// TIA Portal V20 export
// export: Created 2025-12-01T14:57:35.378217Z, ExportSetting None, DisplayName Totally Integrated Automation Portal, DisplayVersion V20 Update 3, DisplayName TIA Portal Openness, DisplayVersion V20 Update 3, DisplayName TIA Portal Version Control Interface, DisplayVersion V20 Update 3, DisplayName STEP 7 Professional, DisplayVersion V20 Update 3, DisplayName STEP 7 Safety, DisplayVersion V20 Update 2, DisplayName WinCC Basic/Comfort/Advanced, DisplayVersion V20 Update 3, DisplayName WinCC Professional, DisplayVersion V20 Update 3, DisplayName WinCC Unified, DisplayVersion V20 Update 3
FUNCTION_BLOCK "FB532_Ordenes_ELEV / VTD_V2"   // FB532, LAD
{ S7_Optimized_Access := 'FALSE' }
// stored: AutoNumber false, SetENOAutomatically false
   VAR_INPUT
      Estado_CBx : "EstadoZona";   // Estado de la Zona
      Maquina { ExternalVisible := 'False'; ExternalWritable := 'False'} : UInt;   // Numero de Máquina
      OrdenDesCarga_OK : Bool;
      Error_Tx : Bool;
   END_VAR
   VAR_OUTPUT
      PosicionDestino : Real;
      Orden : Bool;
   END_VAR
   VAR
      OrdenH01_TipoMovi { ExternalAccessible := 'False'; ExternalVisible := 'False'; ExternalWritable := 'False'; S7_SetPoint := 'True'} : "UDT_VTD_Orden";   // Tipo de Movimiento a Ejecutar con la Horquilla 1
      OrdenH02_TipoMovi { ExternalAccessible := 'False'; ExternalVisible := 'False'; ExternalWritable := 'False'; S7_SetPoint := 'True'} : "UDT_VTD_Orden";   // Tipo de Movimiento a Ejecutar con la Horquilla 2
      OrdenEnCurso : Struct
         EnH01_Poscicion : Real;
         EnH02_Poscicion : Real;
         EnH01_MesaCarga : UInt;
         EnH02_MesaCarga : UInt;
         EnH01_MesaDesCarga : UInt;
         EnH02_MesaDesCarga : UInt;
         EnH01_Existe : Bool;
         EnH02_Existe : Bool;
      END_STRUCT;
      OrdenJdT { ExternalAccessible := 'False'; ExternalVisible := 'False'; ExternalWritable := 'False'} : Struct
         Operacion : UInt;
         MesaHorquilla : UInt;
         MesaCargaDesCarga : UInt;
         VarMesaHorquilla : UInt;
         VarMesaCargaDesCarga : UInt;
         OrdenPoscionado_NOK : Bool;
      END_STRUCT;
      OrdenHMI : Struct
         MesaHorquilla { ExternalAccessible := 'False'; ExternalVisible := 'False'; ExternalWritable := 'False'} : UInt;
         MesaDestino { ExternalAccessible := 'False'; ExternalVisible := 'False'; ExternalWritable := 'False'} : UInt;
         VarMesaHorquilla { ExternalAccessible := 'False'; ExternalVisible := 'False'; ExternalWritable := 'False'} : UInt;
         VarMesaDestino { ExternalAccessible := 'False'; ExternalVisible := 'False'; ExternalWritable := 'False'} : UInt;
      END_STRUCT;
      MemoFlancos { ExternalAccessible := 'False'; ExternalVisible := 'False'; ExternalWritable := 'False'} : Struct
         H1 : Struct
            Posicionar : Bool;
            Carga_E1 : Bool;
            Carga_E2 : Bool;
            Carga_E3 : Bool;
            Carga_E4 : Bool;
            DesCarga_S1 : Bool;
            DesCarga_S2 : Bool;
            DesCarga_S3 : Bool;
            DesCarga_S4 : Bool;
         END_STRUCT;
         H2 : Struct
            Posicionar : Bool;
            Carga_E1 : Bool;
            Carga_E2 : Bool;
            Carga_E3 : Bool;
            Carga_E4 : Bool;
            DesCarga_S1 : Bool;
            DesCarga_S2 : Bool;
            DesCarga_S3 : Bool;
            DesCarga_S4 : Bool;
         END_STRUCT;
      END_STRUCT;
      Peticion : Struct
         Posicion : Real;
         Activa { ExternalAccessible := 'False'; ExternalVisible := 'False'; ExternalWritable := 'False'} : Bool;
      END_STRUCT;
      MesaCargaH01_OK : Bool;
      MesaDesCargaH01_OK : Bool;
      MesaCargaH02_OK : Bool;
      MesaDesCargaH02_OK : Bool;
   END_VAR
   VAR_TEMP
      EstadoVI_VTD : "EstadoMaquina";
      EstadoVI_MesaH1 : "EstadosMesa";   // Estado VI de la Mesa de la H01
      EstadoVI_MesaH2 : "EstadosMesa";   // Estado VI de la Mesa de la H02
      VarUTs : Struct
         PrimeraUT_EnMesa : UInt;
         MesaDestino : UInt;
      END_STRUCT;
      VarBusqueda : Struct
         Posicion : Real;
         Destino : UInt;
         Indice : UInt;
      END_STRUCT;
      VarInterlock : Struct
         Posicion : Real;
         Indice : UInt;
      END_STRUCT;
      NumVTD : UInt;
      NumMesaH1 : UInt;
      NumMesaH2 : UInt;
      Cero : Byte;
      ValorReturn : Int;
      EnMarchaVTDC : Bool;
   END_VAR
   VAR_TEMP   // added for the SCL form of the ladder/FBD networks
      _w1 : Bool;
      _w2 : Bool;
   END_VAR
BEGIN

REGION Network 1 (SCL): Inicializacion
   /////////////////////////////////////////////////////////////////////////////
   // --- Inicializar las Variables
   #Cero := 0;


   /////////////////////////////////////////////////////////////////////////////
   // --- Inicializar Variables En Horquilla 01
   IF #OrdenEnCurso.EnH01_Existe = FALSE THEN
       #ValorReturn := FILL(BVAL := #Cero, BLK => #OrdenH01_TipoMovi);
       #OrdenEnCurso.EnH01_Poscicion := 0.0;
       #OrdenEnCurso.EnH01_MesaCarga := 0;
       #OrdenEnCurso.EnH01_MesaDesCarga := 0;

   END_IF;


   /////////////////////////////////////////////////////////////////////////////
   // --- Inicializar Variables En Horquilla 01
   IF #OrdenEnCurso.EnH02_Existe = FALSE THEN
       #ValorReturn := FILL(BVAL := #Cero, BLK => #OrdenH02_TipoMovi);
       #OrdenEnCurso.EnH02_Poscicion := 0.0;
       #OrdenEnCurso.EnH02_MesaCarga := 0;
       #OrdenEnCurso.EnH02_MesaDesCarga := 0;

   END_IF;
END_REGION

REGION Network 2: ---- En Marcha VTDC
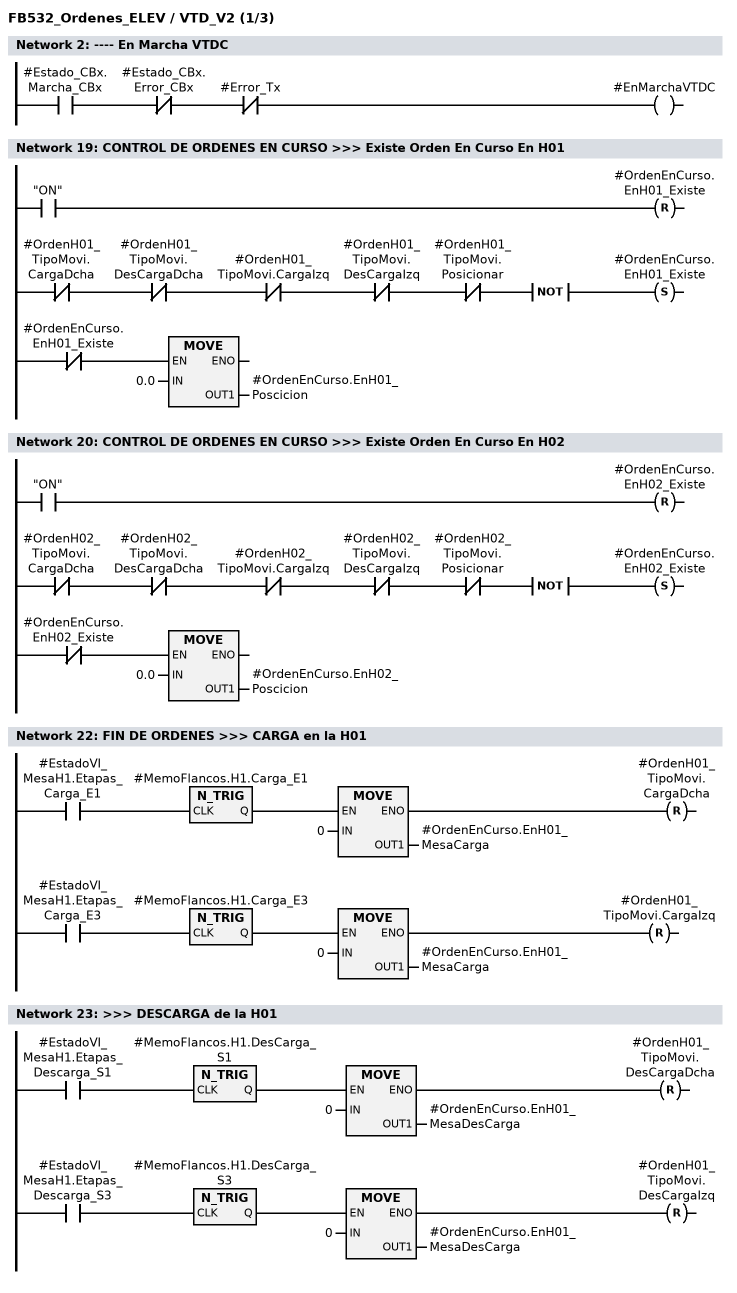
   RUNG wire#powerrail
      Contact( #Estado_CBx.Marcha_CBx )
      I_Contact( #Estado_CBx.Error_CBx )
      I_Contact( #Error_Tx )
      Coil( #EnMarchaVTDC )
   END_RUNG
   // the same network as SCL:
   #EnMarchaVTDC := #Estado_CBx.Marcha_CBx AND NOT #Estado_CBx.Error_CBx AND NOT #Error_Tx;
END_REGION

REGION Network 3 (SCL): ---- Recoger datos de la Maquina
   /////////////////////////////////////////////////////////////////////////////
   // Configuracion 
   #NumMesaH1 := #NumVTD := "DB885_ConfigMaquinas".Maquina[#Maquina].Mesa_1;
   #NumMesaH2 := "DB885_ConfigMaquinas".Maquina[#Maquina].Mesa_2;


   /////////////////////////////////////////////////////////////////////////////
   // Recoger ordenes de JdT
   #OrdenJdT.Operacion := "DB832_Maquinas".Maquinas[#NumVTD].VTD_ELEV.Operacion;
   #OrdenJdT.MesaHorquilla := "DB832_Maquinas".Maquinas[#NumVTD].VTD_ELEV.MesaHorquilla;
   #OrdenJdT.MesaCargaDesCarga := "DB832_Maquinas".Maquinas[#NumVTD].VTD_ELEV.MesaCargaDesCarga;
END_REGION

REGION Network 4 (SCL): ---- Recoger Estado VI de las Horquillas
   /////////////////////////////////////////////////////////////////////////////
   // - Recoger Estado de las Horquillas
   #EstadoVI_VTD := "DB904_Estado_Maquinas".EstadoVI[#NumVTD];
   #EstadoVI_MesaH1 := "DB900_Estado_Mesas".EstadoVI[#NumMesaH1];
   IF #NumMesaH2 <> 0 THEN
       #EstadoVI_MesaH2 := "DB900_Estado_Mesas".EstadoVI[#NumMesaH2];
   ELSE
       #ValorReturn := FILL(BVAL := #Cero, BLK => #EstadoVI_MesaH2);
   END_IF;
END_REGION

REGION Network 5 (SCL): ---- Recoger Variables Internas de las Horquillas
   /////////////////////////////////////////////////////////////////////////////
   // Recoger Variables para la Horquillla 01
   // OrdenDesCarga_OK >>> Permiso para Generar Orden de DesCarga, por si hay que hacer algun Calculo Previo de la Posicion
   #MesaCargaH01_OK := (#EstadoVI_MesaH1.Etapa_Vacia = TRUE) OR (#EstadoVI_MesaH1.Etapas_Descarga_S1 = TRUE) OR (#EstadoVI_MesaH1.Etapas_Descarga_S3 = TRUE);
   #MesaDesCargaH01_OK := (#EstadoVI_MesaH1.Etapa_Cargada = TRUE) AND (#OrdenDesCarga_OK = TRUE);


   /////////////////////////////////////////////////////////////////////////////
   /////////////////////////////////////////////////////////////////////////////
   // Recoger Variables para la Horquillla 02
   IF (#NumMesaH2 <> 0) THEN
       #MesaCargaH02_OK := (#EstadoVI_MesaH2.Etapa_Vacia = TRUE) OR (#EstadoVI_MesaH2.Etapas_Descarga_S1 = TRUE) OR (#EstadoVI_MesaH2.Etapas_Descarga_S3 = TRUE);
       #MesaDesCargaH02_OK := (#EstadoVI_MesaH2.Etapa_Cargada = TRUE);

   ELSE
       #MesaCargaH02_OK := #MesaDesCargaH02_OK = FALSE;

   END_IF;
END_REGION

REGION Network 6 (SCL): ---- Reset de Variables
   /////////////////////////////////////////////////////////////////////////////
   // Reseteo desde JdT
   IF #Estado_CBx.PerReset_CBx = TRUE THEN
       #Peticion.Activa := FALSE;
       #ValorReturn := FILL(BVAL := #Cero, BLK => #OrdenH01_TipoMovi);
       #ValorReturn := FILL(BVAL := #Cero, BLK => #OrdenH02_TipoMovi);

       #OrdenEnCurso.EnH01_Existe := #OrdenEnCurso.EnH02_Existe := FALSE;
       #OrdenEnCurso.EnH01_Poscicion := #OrdenEnCurso.EnH02_Poscicion := 0.0;
       #OrdenEnCurso.EnH01_MesaCarga := #OrdenEnCurso.EnH02_MesaCarga := 0;
       #OrdenEnCurso.EnH01_MesaDesCarga := #OrdenEnCurso.EnH02_MesaDesCarga := 0;

       #Peticion.Activa := FALSE;

   END_IF;
END_REGION

REGION Network 7: >>>>>>>>>>>>>>>>>>>>>>>>>>>>>>>>>>>>>>>>>>>>>>>>>>>>>>>>>>>>>>>>>>>>>>>>>>>>>>>>
END_REGION

REGION Network 8 (SCL): VTDC Doble (Particular del Tipo de Maquina) - Control H01 >>> CARGA
   /////////////////////////////////////////////////////////////////////////////
   // --- CONTROL DE CARGA de la Horquilla 01
   // 
   // --- Esta en Marcha 
   // --- Esta Preparado para Cargar
   // --- Comprobar que no exista Orden En Curso De Carga 
   IF (#EnMarchaVTDC = TRUE) AND (#MesaCargaH01_OK = TRUE) AND
       (#OrdenH01_TipoMovi.CargaDcha = FALSE) AND (#OrdenH01_TipoMovi.CargaIzq = FALSE) AND (#OrdenH01_TipoMovi.Posicionar = FALSE) THEN

       // >>>>> Sin Orden en Curso en la Horquilla 1
       //       Sin Orden En Curso en la Horquilla 2
       IF (#OrdenEnCurso.EnH01_Existe = FALSE) AND (#OrdenEnCurso.EnH02_Existe = FALSE) AND (#Peticion.Posicion = 0) THEN

           FOR #VarBusqueda.Indice := 1 TO "CTE_MaxMesas" DO
               // --- Hay Aviso de Entrada ???
               IF ("DB951_InterlockMaquinas".Maquina[#Maquina].Mesa[#VarBusqueda.Indice].Out.AVTF = TRUE) THEN

                   ////////////////////////////////////////////////////////////////////////////////
                   // --- Es Destino la Horquilla
                   #VarUTs.PrimeraUT_EnMesa := "DB810_ColasMesas".Colas[#VarBusqueda.Indice].UT_PrimeraMesa;
                   #VarBusqueda.Destino := "DB812_UTs_Control".UT[#VarUTs.PrimeraUT_EnMesa].MesaDestino;
                   #VarBusqueda.Destino := #VarBusqueda.Destino - "CTE_OffsetMesa";
                   IF (#VarBusqueda.Destino = #NumMesaH1) THEN
                       ////////////////////////////////////////////////////////////////////////////////
                       // --- Es En Carga Derecha
                       IF "DB885_ConfigMaquinas".Maquina[#Maquina].Mesa[#VarBusqueda.Indice].Derecha = TRUE THEN
                           #OrdenEnCurso.EnH01_Poscicion := "DB885_ConfigMaquinas".Maquina[#Maquina].Mesa[#VarBusqueda.Indice].Posicion_mm_H1;
                           #OrdenEnCurso.EnH01_MesaCarga := #VarBusqueda.Indice;
                           #OrdenH01_TipoMovi.CargaDcha := TRUE;
                           #OrdenEnCurso.EnH01_Existe := TRUE;
                           EXIT;
                       END_IF;
                       ////////////////////////////////////////////////////////////////////////////////
                       // --- Es En Carga Izquierda
                       IF "DB885_ConfigMaquinas".Maquina[#Maquina].Mesa[#VarBusqueda.Indice].Izquierda = TRUE THEN
                           #OrdenEnCurso.EnH01_Poscicion := "DB885_ConfigMaquinas".Maquina[#Maquina].Mesa[#VarBusqueda.Indice].Posicion_mm_H1;
                           #OrdenEnCurso.EnH01_MesaCarga := #VarBusqueda.Indice;
                           #OrdenH01_TipoMovi.CargaIzq := TRUE;
                           #OrdenEnCurso.EnH01_Existe := TRUE;
                           EXIT;
                       END_IF;
                   END_IF;
                   ////////////////////////////////////////////////////////////////////////////////

               END_IF;
           END_FOR;

       END_IF;


       // >>>>> Sin Orden en Curso en la Horquilla 1
       //       Con Orden En Curso en la Horquilla 2
       IF #OrdenEnCurso.EnH01_Existe = FALSE AND #OrdenEnCurso.EnH02_Existe = TRUE THEN
           #VarBusqueda.Posicion := #Peticion.Posicion;

           FOR #VarBusqueda.Indice := 1 TO "CTE_MaxMesas" DO
               // --- Hay Aviso de Entrada ???
               IF ("DB951_InterlockMaquinas".Maquina[#Maquina].Mesa[#VarBusqueda.Indice].Out.AVTF = TRUE) AND
                   ("DB885_ConfigMaquinas".Maquina[#Maquina].Mesa[#VarBusqueda.Indice].Posicion_mm_H1 = #VarBusqueda.Posicion) THEN

                   ////////////////////////////////////////////////////////////////////////////////
                   // --- Es Destino la Horquilla
                   #VarUTs.PrimeraUT_EnMesa := "DB810_ColasMesas".Colas[#VarBusqueda.Indice].UT_PrimeraMesa;
                   #VarBusqueda.Destino := "DB812_UTs_Control".UT[#VarUTs.PrimeraUT_EnMesa].MesaDestino;
                   #VarBusqueda.Destino := #VarBusqueda.Destino - "CTE_OffsetMesa";
                   IF (#VarBusqueda.Destino = #NumMesaH1) THEN
                       ////////////////////////////////////////////////////////////////////////////////
                       // --- Es En Carga Derecha
                       IF ("DB885_ConfigMaquinas".Maquina[#Maquina].Mesa[#VarBusqueda.Indice].Derecha = TRUE) THEN
                           #OrdenEnCurso.EnH01_Poscicion := "DB885_ConfigMaquinas".Maquina[#Maquina].Mesa[#VarBusqueda.Indice].Posicion_mm_H1;
                           #OrdenEnCurso.EnH01_MesaCarga := #VarBusqueda.Indice;
                           #OrdenH01_TipoMovi.CargaDcha := TRUE;
                           #OrdenEnCurso.EnH01_Existe := TRUE;
                           EXIT;
                       END_IF;
                       ////////////////////////////////////////////////////////////////////////////////
                       // --- Es En Carga Izquierda
                       IF ("DB885_ConfigMaquinas".Maquina[#Maquina].Mesa[#VarBusqueda.Indice].Izquierda = TRUE) THEN
                           #OrdenEnCurso.EnH01_Poscicion := "DB885_ConfigMaquinas".Maquina[#Maquina].Mesa[#VarBusqueda.Indice].Posicion_mm_H1;
                           #OrdenEnCurso.EnH01_MesaCarga := #VarBusqueda.Indice;
                           #OrdenH01_TipoMovi.CargaIzq := TRUE;
                           #OrdenEnCurso.EnH01_Existe := TRUE;
                           EXIT;
                       END_IF;
                   END_IF;
                   ////////////////////////////////////////////////////////////////////////////////

               END_IF;
           END_FOR;

       END_IF;


       // >>>>> Con Orden en Curso en la Horquilla 1
       //       Sin o Con Orden En Curso en la Horquilla 2
       IF #OrdenEnCurso.EnH01_Existe = TRUE THEN
           #VarBusqueda.Posicion := #Peticion.Posicion;

           FOR #VarBusqueda.Indice := 1 TO "CTE_MaxMesas" DO
               // --- Hay Aviso de Entrada ???
               IF ("DB951_InterlockMaquinas".Maquina[#Maquina].Mesa[#VarBusqueda.Indice].Out.AVTF = TRUE) AND
                   ("DB885_ConfigMaquinas".Maquina[#Maquina].Mesa[#VarBusqueda.Indice].Posicion_mm_H1 = #VarBusqueda.Posicion) THEN

                   ////////////////////////////////////////////////////////////////////////////////
                   // --- Es Destino la Horquilla
                   #VarUTs.PrimeraUT_EnMesa := "DB810_ColasMesas".Colas[#VarBusqueda.Indice].UT_PrimeraMesa;
                   #VarBusqueda.Destino := "DB812_UTs_Control".UT[#VarUTs.PrimeraUT_EnMesa].MesaDestino;
                   #VarBusqueda.Destino := #VarBusqueda.Destino - "CTE_OffsetMesa";
                   IF (#VarBusqueda.Destino = #NumMesaH1) THEN
                       ////////////////////////////////////////////////////////////////////////////////
                       // --- Es En Carga Derecha
                       IF ("DB885_ConfigMaquinas".Maquina[#Maquina].Mesa[#VarBusqueda.Indice].Derecha = TRUE) AND (#OrdenH01_TipoMovi.DesCargaIzq = TRUE) THEN
                           #OrdenEnCurso.EnH01_Poscicion := "DB885_ConfigMaquinas".Maquina[#Maquina].Mesa[#VarBusqueda.Indice].Posicion_mm_H1;
                           #OrdenEnCurso.EnH01_MesaCarga := #VarBusqueda.Indice;
                           #OrdenH01_TipoMovi.CargaDcha := TRUE;
                           #OrdenEnCurso.EnH01_Existe := TRUE;
                           EXIT;
                       END_IF;
                       ////////////////////////////////////////////////////////////////////////////////
                       // --- Es En Carga Izquierda
                       IF ("DB885_ConfigMaquinas".Maquina[#Maquina].Mesa[#VarBusqueda.Indice].Izquierda = TRUE) AND (#OrdenH01_TipoMovi.DesCargaDcha = TRUE) THEN
                           #OrdenEnCurso.EnH01_Poscicion := "DB885_ConfigMaquinas".Maquina[#Maquina].Mesa[#VarBusqueda.Indice].Posicion_mm_H1;
                           #OrdenEnCurso.EnH01_MesaCarga := #VarBusqueda.Indice;
                           #OrdenH01_TipoMovi.CargaIzq := TRUE;
                           #OrdenEnCurso.EnH01_Existe := TRUE;
                           EXIT;
                       END_IF;
                   END_IF;
                   ////////////////////////////////////////////////////////////////////////////////

               END_IF;
           END_FOR;

       END_IF;

   END_IF;
END_REGION

REGION Network 9 (SCL): VTDC Doble (Particular del Tipo de Maquina) - Control H01 >>> DESCARGA
   /////////////////////////////////////////////////////////////////////////////
   // --- CONTROL DE DESCARGA de la Horquilla 01
   // 
   // --- Esta en Marcha 
   // --- Esta Preparado para Cargar
   // --- Comprobar que no exista Orden En Curso De DesCarga 
   IF (#EnMarchaVTDC = TRUE) AND (#MesaDesCargaH01_OK = TRUE) AND
       (#OrdenH01_TipoMovi.DesCargaDcha = FALSE) AND (#OrdenH01_TipoMovi.DesCargaIzq = FALSE) AND (#OrdenH01_TipoMovi.Posicionar = FALSE) THEN

       /////////////////////////////////////////////////////////////////////////////
       // --- Recoger Destino de UT 
       #VarUTs.MesaDestino := 0;
       #VarUTs.PrimeraUT_EnMesa := "DB810_ColasMesas".Colas[#NumMesaH1].UT_PrimeraMesa;
       IF #VarUTs.PrimeraUT_EnMesa <> 0 THEN
           #VarUTs.MesaDestino := "DB812_UTs_Control".UT[#VarUTs.PrimeraUT_EnMesa].MesaDestino;
           IF (#VarUTs.MesaDestino <> 0) THEN
               #VarUTs.MesaDestino := #VarUTs.MesaDestino - "CTE_OffsetMesa";
               IF (#VarUTs.MesaDestino = #NumMesaH1) THEN
                   #VarUTs.MesaDestino := 0;
               END_IF;
           END_IF;

       END_IF;

       /////////////////////////////////////////////////////////////////////////////
       // --- Existe Destino de Salida
       IF #VarUTs.MesaDestino <> 0 THEN

           /////////////////////////////////////////////////////////////////////////////
           // >>>>> Sin Orden en Curso en la Horquilla 1
           //       Sin Orden En Curso en la Horquilla 2
           IF (#OrdenEnCurso.EnH01_Existe = FALSE) AND (#OrdenEnCurso.EnH02_Existe = FALSE) AND (#Peticion.Posicion = 0) THEN

               ////////////////////////////////////////////////////////////////////////////////
               // --- Es En DesCarga Derecha
               IF ("DB885_ConfigMaquinas".Maquina[#Maquina].Mesa[#VarUTs.MesaDestino].Derecha = TRUE) THEN
                   #OrdenEnCurso.EnH01_Poscicion := "DB885_ConfigMaquinas".Maquina[#Maquina].Mesa[#VarUTs.MesaDestino].Posicion_mm_H1;
                   #OrdenEnCurso.EnH01_MesaDesCarga := #VarUTs.MesaDestino;
                   #OrdenH01_TipoMovi.DesCargaDcha := TRUE;
                   #OrdenEnCurso.EnH01_Existe := TRUE;

               END_IF;
               ////////////////////////////////////////////////////////////////////////////////
               // --- Es En DesCarga Izquierda
               IF ("DB885_ConfigMaquinas".Maquina[#Maquina].Mesa[#VarUTs.MesaDestino].Izquierda = TRUE) THEN
                   #OrdenEnCurso.EnH01_Poscicion := "DB885_ConfigMaquinas".Maquina[#Maquina].Mesa[#VarUTs.MesaDestino].Posicion_mm_H1;
                   #OrdenEnCurso.EnH01_MesaDesCarga := #VarUTs.MesaDestino;
                   #OrdenH01_TipoMovi.DesCargaIzq := TRUE;
                   #OrdenEnCurso.EnH01_Existe := TRUE;

               END_IF;
               ////////////////////////////////////////////////////////////////////////////////

           END_IF;

           /////////////////////////////////////////////////////////////////////////////
           // >>>>> Sin Orden en Curso en la Horquilla 1
           //       Con Orden En Curso en la Horquilla 2
           IF (#OrdenEnCurso.EnH01_Existe = FALSE) AND (#OrdenEnCurso.EnH02_Existe = TRUE) THEN
               #VarBusqueda.Posicion := #Peticion.Posicion;

               // >>> Esta En Posicion Actual 
               IF ("DB885_ConfigMaquinas".Maquina[#Maquina].Mesa[#VarUTs.MesaDestino].Posicion_mm_H1 = #VarBusqueda.Posicion) THEN

                   ////////////////////////////////////////////////////////////////////////////////
                   // --- Es En DesCarga Derecha
                   IF ("DB885_ConfigMaquinas".Maquina[#Maquina].Mesa[#VarUTs.MesaDestino].Derecha = TRUE) THEN
                       #OrdenEnCurso.EnH01_Poscicion := "DB885_ConfigMaquinas".Maquina[#Maquina].Mesa[#VarUTs.MesaDestino].Posicion_mm_H1;
                       #OrdenEnCurso.EnH01_MesaDesCarga := #VarUTs.MesaDestino;
                       #OrdenH01_TipoMovi.DesCargaDcha := TRUE;
                       #OrdenEnCurso.EnH01_Existe := TRUE;

                   END_IF;
                   ////////////////////////////////////////////////////////////////////////////////
                   // --- Es En DesCarga Izquierda
                   IF ("DB885_ConfigMaquinas".Maquina[#Maquina].Mesa[#VarUTs.MesaDestino].Izquierda = TRUE) THEN
                       #OrdenEnCurso.EnH01_Poscicion := "DB885_ConfigMaquinas".Maquina[#Maquina].Mesa[#VarUTs.MesaDestino].Posicion_mm_H1;
                       #OrdenEnCurso.EnH01_MesaDesCarga := #VarUTs.MesaDestino;
                       #OrdenH01_TipoMovi.DesCargaIzq := TRUE;
                       #OrdenEnCurso.EnH01_Existe := TRUE;

                   END_IF;
                   ////////////////////////////////////////////////////////////////////////////////

               END_IF;
           END_IF;

           /////////////////////////////////////////////////////////////////////////////
           // >>>>> Con Orden en Curso en la Horquilla 1
           //       Sin y Con Orden En Curso en la Horquilla 2
           IF (#OrdenEnCurso.EnH01_Existe = TRUE) THEN
               #VarBusqueda.Posicion := #Peticion.Posicion;

               // >>> Esta En Posicion Actual 
               IF ("DB885_ConfigMaquinas".Maquina[#Maquina].Mesa[#VarUTs.MesaDestino].Posicion_mm_H1 = #VarBusqueda.Posicion) THEN

                   ////////////////////////////////////////////////////////////////////////////////
                   // --- Es En DesCarga Derecha
                   IF ("DB885_ConfigMaquinas".Maquina[#Maquina].Mesa[#VarUTs.MesaDestino].Derecha = TRUE) AND (#OrdenH01_TipoMovi.CargaIzq = TRUE)  THEN
                       #OrdenEnCurso.EnH01_Poscicion := "DB885_ConfigMaquinas".Maquina[#Maquina].Mesa[#VarUTs.MesaDestino].Posicion_mm_H1;
                       #OrdenEnCurso.EnH01_MesaDesCarga := #VarUTs.MesaDestino;
                       #OrdenH01_TipoMovi.DesCargaDcha := TRUE;
                       #OrdenEnCurso.EnH01_Existe := TRUE;

                   END_IF;
                   ////////////////////////////////////////////////////////////////////////////////
                   // --- Es En DesCarga Izquierda
                   IF ("DB885_ConfigMaquinas".Maquina[#Maquina].Mesa[#VarUTs.MesaDestino].Izquierda = TRUE) AND (#OrdenH01_TipoMovi.CargaDcha = TRUE) THEN
                       #OrdenEnCurso.EnH01_Poscicion := "DB885_ConfigMaquinas".Maquina[#Maquina].Mesa[#VarUTs.MesaDestino].Posicion_mm_H1;
                       #OrdenEnCurso.EnH01_MesaDesCarga := #VarUTs.MesaDestino;
                       #OrdenH01_TipoMovi.DesCargaIzq := TRUE;
                       #OrdenEnCurso.EnH01_Existe := TRUE;

                   END_IF;
                   ////////////////////////////////////////////////////////////////////////////////

               END_IF;
           END_IF;
       END_IF;

   END_IF;
END_REGION

REGION Network 10: >>>>>>>>>>>>>>>>>>>>>>>>>>>>>>>>>>>>>>>>>>>>>>>>>>>>>>>>>>>>>>>>>>>>>>>>>>>>>>>>
END_REGION

REGION Network 11 (SCL): VTDC Doble (Particular del Tipo de Maquina) - Control H02 >>> CARGA
   /////////////////////////////////////////////////////////////////////////////
   // --- CONTROL DE CARGA de la Horquilla 01
   // 
   // --- Esta en Marcha 
   // --- Esta Preparado para Cargar
   // --- Comprobar que no exista Orden En Curso De Carga 
   IF (#EnMarchaVTDC = TRUE) AND (#MesaCargaH02_OK = TRUE) AND
       (#OrdenH02_TipoMovi.CargaDcha = FALSE) AND (#OrdenH02_TipoMovi.CargaIzq = FALSE) AND (#OrdenH02_TipoMovi.Posicionar = FALSE) THEN

       // >>>>> Sin Orden en Curso en la Horquilla 1
       //       Sin Orden En Curso en la Horquilla 2
       IF (#OrdenEnCurso.EnH01_Existe = FALSE) AND (#OrdenEnCurso.EnH02_Existe = FALSE) AND (#Peticion.Posicion = 0) THEN

           FOR #VarBusqueda.Indice := 1 TO "CTE_MaxMesas" DO
               // --- Hay Aviso de Entrada ???
               IF ("DB951_InterlockMaquinas".Maquina[#Maquina].Mesa[#VarBusqueda.Indice].Out.AVTF = TRUE) THEN

                   ////////////////////////////////////////////////////////////////////////////////
                   // --- Es Destino la Horquilla
                   #VarUTs.PrimeraUT_EnMesa := "DB810_ColasMesas".Colas[#VarBusqueda.Indice].UT_PrimeraMesa;
                   #VarBusqueda.Destino := "DB812_UTs_Control".UT[#VarUTs.PrimeraUT_EnMesa].MesaDestino;
                   #VarBusqueda.Destino := #VarBusqueda.Destino - "CTE_OffsetMesa";
                   IF (#VarBusqueda.Destino = #NumMesaH2) THEN
                       ////////////////////////////////////////////////////////////////////////////////
                       // --- Es En Carga Derecha
                       IF "DB885_ConfigMaquinas".Maquina[#Maquina].Mesa[#VarBusqueda.Indice].Derecha = TRUE THEN
                           #OrdenEnCurso.EnH02_Poscicion := "DB885_ConfigMaquinas".Maquina[#Maquina].Mesa[#VarBusqueda.Indice].Posicion_mm_H2;
                           #OrdenEnCurso.EnH02_MesaCarga := #VarBusqueda.Indice;
                           #OrdenH02_TipoMovi.CargaDcha := TRUE;
                           #OrdenEnCurso.EnH02_Existe := TRUE;
                           EXIT;
                       END_IF;
                       ////////////////////////////////////////////////////////////////////////////////
                       // --- Es En Carga Izquierda
                       IF "DB885_ConfigMaquinas".Maquina[#Maquina].Mesa[#VarBusqueda.Indice].Izquierda = TRUE THEN
                           #OrdenEnCurso.EnH02_Poscicion := "DB885_ConfigMaquinas".Maquina[#Maquina].Mesa[#VarBusqueda.Indice].Posicion_mm_H2;
                           #OrdenEnCurso.EnH02_MesaCarga := #VarBusqueda.Indice;
                           #OrdenH02_TipoMovi.CargaIzq := TRUE;
                           #OrdenEnCurso.EnH02_Existe := TRUE;
                           EXIT;
                       END_IF;
                   END_IF;
                   ////////////////////////////////////////////////////////////////////////////////

               END_IF;
           END_FOR;

       END_IF;


       // >>>>> Con Orden en Curso en la Horquilla 1
       //       Sin Orden En Curso en la Horquilla 2
       IF #OrdenEnCurso.EnH01_Existe = TRUE AND #OrdenEnCurso.EnH02_Existe = FALSE THEN
           #VarBusqueda.Posicion := #Peticion.Posicion;

           FOR #VarBusqueda.Indice := 1 TO "CTE_MaxMesas" DO
               // --- Hay Aviso de Entrada ???
               IF ("DB951_InterlockMaquinas".Maquina[#Maquina].Mesa[#VarBusqueda.Indice].Out.AVTF = TRUE) AND
                   ("DB885_ConfigMaquinas".Maquina[#Maquina].Mesa[#VarBusqueda.Indice].Posicion_mm_H2 = #VarBusqueda.Posicion) THEN

                   ////////////////////////////////////////////////////////////////////////////////
                   // --- Es Destino la Horquilla
                   #VarUTs.PrimeraUT_EnMesa := "DB810_ColasMesas".Colas[#VarBusqueda.Indice].UT_PrimeraMesa;
                   #VarBusqueda.Destino := "DB812_UTs_Control".UT[#VarUTs.PrimeraUT_EnMesa].MesaDestino;
                   #VarBusqueda.Destino := #VarBusqueda.Destino - "CTE_OffsetMesa";
                   IF (#VarBusqueda.Destino = #NumMesaH2) THEN
                       ////////////////////////////////////////////////////////////////////////////////
                       // --- Es En Carga Derecha
                       IF ("DB885_ConfigMaquinas".Maquina[#Maquina].Mesa[#VarBusqueda.Indice].Derecha = TRUE) THEN
                           #OrdenEnCurso.EnH02_Poscicion := "DB885_ConfigMaquinas".Maquina[#Maquina].Mesa[#VarBusqueda.Indice].Posicion_mm_H2;
                           #OrdenEnCurso.EnH02_MesaCarga := #VarBusqueda.Indice;
                           #OrdenH02_TipoMovi.CargaDcha := TRUE;
                           #OrdenEnCurso.EnH02_Existe := TRUE;
                           EXIT;
                       END_IF;
                       ////////////////////////////////////////////////////////////////////////////////
                       // --- Es En Carga Izquierda
                       IF ("DB885_ConfigMaquinas".Maquina[#Maquina].Mesa[#VarBusqueda.Indice].Izquierda = TRUE) THEN
                           #OrdenEnCurso.EnH02_Poscicion := "DB885_ConfigMaquinas".Maquina[#Maquina].Mesa[#VarBusqueda.Indice].Posicion_mm_H2;
                           #OrdenEnCurso.EnH02_MesaCarga := #VarBusqueda.Indice;
                           #OrdenH02_TipoMovi.CargaIzq := TRUE;
                           #OrdenEnCurso.EnH02_Existe := TRUE;
                           EXIT;
                       END_IF;
                   END_IF;
                   ////////////////////////////////////////////////////////////////////////////////

               END_IF;
           END_FOR;

       END_IF;


       // >>>>> Sin o Con Orden en Curso en la Horquilla 1
       //       Con Orden En Curso en la Horquilla 2
       IF #OrdenEnCurso.EnH02_Existe = TRUE THEN
           #VarBusqueda.Posicion := #Peticion.Posicion;

           FOR #VarBusqueda.Indice := 1 TO "CTE_MaxMesas" DO
               // --- Hay Aviso de Entrada ???
               IF ("DB951_InterlockMaquinas".Maquina[#Maquina].Mesa[#VarBusqueda.Indice].Out.AVTF = TRUE) AND
                   ("DB885_ConfigMaquinas".Maquina[#Maquina].Mesa[#VarBusqueda.Indice].Posicion_mm_H2 = #VarBusqueda.Posicion) THEN

                   ////////////////////////////////////////////////////////////////////////////////
                   // --- Es Destino la Horquilla 1
                   #VarUTs.PrimeraUT_EnMesa := "DB810_ColasMesas".Colas[#VarBusqueda.Indice].UT_PrimeraMesa;
                   #VarBusqueda.Destino := "DB812_UTs_Control".UT[#VarUTs.PrimeraUT_EnMesa].MesaDestino;
                   #VarBusqueda.Destino := #VarBusqueda.Destino - "CTE_OffsetMesa";
                   IF (#VarBusqueda.Destino = #NumMesaH2) THEN
                       ////////////////////////////////////////////////////////////////////////////////
                       // --- Es En Carga Derecha
                       IF ("DB885_ConfigMaquinas".Maquina[#Maquina].Mesa[#VarBusqueda.Indice].Derecha = TRUE) AND (#OrdenH02_TipoMovi.DesCargaIzq = TRUE) THEN
                           #OrdenEnCurso.EnH02_Poscicion := "DB885_ConfigMaquinas".Maquina[#Maquina].Mesa[#VarBusqueda.Indice].Posicion_mm_H2;
                           #OrdenEnCurso.EnH02_MesaCarga := #VarBusqueda.Indice;
                           #OrdenH02_TipoMovi.CargaDcha := TRUE;
                           #OrdenEnCurso.EnH02_Existe := TRUE;
                           EXIT;
                       END_IF;
                       ////////////////////////////////////////////////////////////////////////////////
                       // --- Es En Carga Izquierda
                       IF ("DB885_ConfigMaquinas".Maquina[#Maquina].Mesa[#VarBusqueda.Indice].Izquierda = TRUE) AND (#OrdenH02_TipoMovi.DesCargaDcha = TRUE) THEN
                           #OrdenEnCurso.EnH02_Poscicion := "DB885_ConfigMaquinas".Maquina[#Maquina].Mesa[#VarBusqueda.Indice].Posicion_mm_H2;
                           #OrdenEnCurso.EnH02_MesaCarga := #VarBusqueda.Indice;
                           #OrdenH02_TipoMovi.CargaIzq := TRUE;
                           #OrdenEnCurso.EnH02_Existe := TRUE;
                           EXIT;
                       END_IF;
                   END_IF;
                   ////////////////////////////////////////////////////////////////////////////////

               END_IF;
           END_FOR;

       END_IF;

   END_IF;
END_REGION

REGION Network 12 (SCL): VTDC Doble (Particular del Tipo de Maquina) - Control H02 >>> DESCARGA
   /////////////////////////////////////////////////////////////////////////////
   // --- CONTROL DE DESCARGA de la Horquilla 02
   // 
   // --- Esta en Marcha 
   // --- Esta Preparado para Cargar
   // --- Comprobar que no exista Orden En Curso De DesCarga 
   IF (#EnMarchaVTDC = TRUE) AND (#MesaDesCargaH02_OK = TRUE) AND
       (#OrdenH02_TipoMovi.DesCargaDcha = FALSE) AND (#OrdenH02_TipoMovi.DesCargaIzq = FALSE) AND (#OrdenH02_TipoMovi.Posicionar = FALSE) THEN

       /////////////////////////////////////////////////////////////////////////////
       // --- Recoger Destino de UT 
       #VarUTs.MesaDestino := 0;
       #VarUTs.PrimeraUT_EnMesa := "DB810_ColasMesas".Colas[#NumMesaH2].UT_PrimeraMesa;
       IF #VarUTs.PrimeraUT_EnMesa <> 0 THEN
           #VarUTs.MesaDestino := "DB812_UTs_Control".UT[#VarUTs.PrimeraUT_EnMesa].MesaDestino;
           IF (#VarUTs.MesaDestino <> 0) THEN
               #VarUTs.MesaDestino := #VarUTs.MesaDestino - "CTE_OffsetMesa";
               IF (#VarUTs.MesaDestino = #NumMesaH2) THEN
                   #VarUTs.MesaDestino := 0;
               END_IF;
           END_IF;

       END_IF;

       /////////////////////////////////////////////////////////////////////////////
       // --- Existe Destino de Salida
       IF #VarUTs.MesaDestino <> 0 THEN

           /////////////////////////////////////////////////////////////////////////////
           // >>>>> Sin Orden en Curso en la Horquilla 1
           //       Sin Orden En Curso en la Horquilla 2
           IF (#OrdenEnCurso.EnH01_Existe = FALSE) AND (#OrdenEnCurso.EnH02_Existe = FALSE) AND (#Peticion.Posicion = 0) THEN

               ////////////////////////////////////////////////////////////////////////////////
               // --- Es En DesCarga Derecha
               IF ("DB885_ConfigMaquinas".Maquina[#Maquina].Mesa[#VarUTs.MesaDestino].Derecha = TRUE) THEN
                   #OrdenEnCurso.EnH02_Poscicion := "DB885_ConfigMaquinas".Maquina[#Maquina].Mesa[#VarUTs.MesaDestino].Posicion_mm_H2;
                   #OrdenEnCurso.EnH02_MesaDesCarga := #VarUTs.MesaDestino;
                   #OrdenH02_TipoMovi.DesCargaDcha := TRUE;
                   #OrdenEnCurso.EnH02_Existe := TRUE;

               END_IF;
               ////////////////////////////////////////////////////////////////////////////////
               // --- Es En DesCarga Izquierda
               IF ("DB885_ConfigMaquinas".Maquina[#Maquina].Mesa[#VarUTs.MesaDestino].Izquierda = TRUE) THEN
                   #OrdenEnCurso.EnH02_Poscicion := "DB885_ConfigMaquinas".Maquina[#Maquina].Mesa[#VarUTs.MesaDestino].Posicion_mm_H2;
                   #OrdenEnCurso.EnH02_MesaDesCarga := #VarUTs.MesaDestino;
                   #OrdenH02_TipoMovi.DesCargaIzq := TRUE;
                   #OrdenEnCurso.EnH02_Existe := TRUE;

               END_IF;
               ////////////////////////////////////////////////////////////////////////////////

           END_IF;

           /////////////////////////////////////////////////////////////////////////////
           // >>>>> Con Orden en Curso en la Horquilla 1
           //       Sin Orden En Curso en la Horquilla 2
           IF (#OrdenEnCurso.EnH01_Existe = TRUE) AND (#OrdenEnCurso.EnH02_Existe = FALSE) THEN
               #VarBusqueda.Posicion := #Peticion.Posicion;

               // >>> Esta En Posicion Actual 
               IF ("DB885_ConfigMaquinas".Maquina[#Maquina].Mesa[#VarUTs.MesaDestino].Posicion_mm_H2 = #VarBusqueda.Posicion) THEN

                   ////////////////////////////////////////////////////////////////////////////////
                   // --- Es En DesCarga Derecha
                   IF ("DB885_ConfigMaquinas".Maquina[#Maquina].Mesa[#VarUTs.MesaDestino].Derecha = TRUE) THEN
                       #OrdenEnCurso.EnH02_Poscicion := "DB885_ConfigMaquinas".Maquina[#Maquina].Mesa[#VarUTs.MesaDestino].Posicion_mm_H2;
                       #OrdenEnCurso.EnH02_MesaDesCarga := #VarUTs.MesaDestino;
                       #OrdenH02_TipoMovi.DesCargaDcha := TRUE;
                       #OrdenEnCurso.EnH02_Existe := TRUE;

                   END_IF;
                   ////////////////////////////////////////////////////////////////////////////////
                   // --- Es En DesCarga Izquierda
                   IF ("DB885_ConfigMaquinas".Maquina[#Maquina].Mesa[#VarUTs.MesaDestino].Izquierda = TRUE) THEN
                       #OrdenEnCurso.EnH02_Poscicion := "DB885_ConfigMaquinas".Maquina[#Maquina].Mesa[#VarUTs.MesaDestino].Posicion_mm_H2;
                       #OrdenEnCurso.EnH02_MesaDesCarga := #VarUTs.MesaDestino;
                       #OrdenH02_TipoMovi.DesCargaIzq := TRUE;
                       #OrdenEnCurso.EnH02_Existe := TRUE;

                   END_IF;
                   ////////////////////////////////////////////////////////////////////////////////

               END_IF;
           END_IF;

           /////////////////////////////////////////////////////////////////////////////
           // >>>>> Sin y Con Orden en Curso en la Horquilla 1
           //       Con Orden En Curso en la Horquilla 2
           IF (#OrdenEnCurso.EnH02_Existe = TRUE) THEN
               #VarBusqueda.Posicion := #Peticion.Posicion;

               // >>> Esta En Posicion Actual 
               IF ("DB885_ConfigMaquinas".Maquina[#Maquina].Mesa[#VarUTs.MesaDestino].Posicion_mm_H2 = #VarBusqueda.Posicion) THEN

                   ////////////////////////////////////////////////////////////////////////////////
                   // --- Es En DesCarga Derecha
                   IF ("DB885_ConfigMaquinas".Maquina[#Maquina].Mesa[#VarUTs.MesaDestino].Derecha = TRUE) AND (#OrdenH02_TipoMovi.CargaIzq = TRUE) THEN
                       #OrdenEnCurso.EnH02_Poscicion := "DB885_ConfigMaquinas".Maquina[#Maquina].Mesa[#VarUTs.MesaDestino].Posicion_mm_H2;
                       #OrdenEnCurso.EnH02_MesaDesCarga := #VarUTs.MesaDestino;
                       #OrdenH02_TipoMovi.DesCargaDcha := TRUE;
                       #OrdenEnCurso.EnH02_Existe := TRUE;

                   END_IF;
                   ////////////////////////////////////////////////////////////////////////////////
                   // --- Es En DesCarga Izquierda
                   IF ("DB885_ConfigMaquinas".Maquina[#Maquina].Mesa[#VarUTs.MesaDestino].Izquierda = TRUE) AND (#OrdenH02_TipoMovi.CargaDcha = TRUE) THEN
                       #OrdenEnCurso.EnH02_Poscicion := "DB885_ConfigMaquinas".Maquina[#Maquina].Mesa[#VarUTs.MesaDestino].Posicion_mm_H2;
                       #OrdenEnCurso.EnH02_MesaDesCarga := #VarUTs.MesaDestino;
                       #OrdenH02_TipoMovi.DesCargaIzq := TRUE;
                       #OrdenEnCurso.EnH02_Existe := TRUE;

                   END_IF;
                   ////////////////////////////////////////////////////////////////////////////////

               END_IF;
           END_IF;
       END_IF;

   END_IF;
END_REGION

REGION Network 13: >>>>>>>>>>>>>>>>>>>>>>>>>>>>>>>>>>>>>>>>>>>>>>>>>>>>>>>>>>>>>>>>>>>>>>>>>>>>>>>>
END_REGION

REGION Network 14 (SCL): JDT >>> Peticion de la Posicion Actual del VTD
   /////////////////////////////////////////////////////////////////////////////
   // --- Peticion de la Posicion Actual del VTD

   IF (#OrdenJdT.Operacion = "CTE_OperacionSTAT") THEN
       IF ("DB832_Maquinas".Maquinas[#NumVTD].VTD_ELEV.Respuesta = 0) THEN
           "DB832_Maquinas".Maquinas[#NumVTD].VTD_ELEV.Respuesta := "Evento_VTDC_PosicionActualVTD";
           "DB832_Maquinas".Maquinas[#NumVTD].VTD_ELEV.Operacion := 0;
           #OrdenJdT.Operacion := 0;
       END_IF;

   END_IF;
END_REGION

REGION Network 15 (SCL): JDT >>> Orden de Posicionar el VTD (Horquilla, Mesa Carga o DesCarga)
   /////////////////////////////////////////////////////////////////////////////
   // --- Orden de Posicionar el VTD (Horquilla, Mesa Carga o DesCarga)

   IF (#OrdenJdT.Operacion = "CTE_OperacionPOSI") AND (#OrdenJdT.MesaHorquilla <> 0) AND (#OrdenJdT.MesaCargaDesCarga <> 0) AND
       (#EnMarchaVTDC = TRUE) AND (#OrdenEnCurso.EnH01_Existe = FALSE) AND (#OrdenEnCurso.EnH02_Existe = FALSE) THEN
       #OrdenJdT.VarMesaHorquilla := #OrdenJdT.MesaHorquilla - "CTE_OffsetMesa";
       #OrdenJdT.VarMesaCargaDesCarga := #OrdenJdT.MesaCargaDesCarga - "CTE_OffsetMesa";
       #OrdenJdT.OrdenPoscionado_NOK := FALSE;

       //////////////////////////////////////////////////////////////////////
       // Orden de Posicionar a la Horquilla 1
       IF (#OrdenJdT.VarMesaHorquilla = #NumMesaH1) THEN
           IF ("DB885_ConfigMaquinas".Maquina[#Maquina].Mesa[#OrdenJdT.VarMesaCargaDesCarga].Posicion_mm_H1 <> 0) THEN
               #OrdenEnCurso.EnH01_Poscicion := "DB885_ConfigMaquinas".Maquina[#Maquina].Mesa[#OrdenJdT.VarMesaCargaDesCarga].Posicion_mm_H1;
               #OrdenH01_TipoMovi.Posicionar := TRUE;
               #OrdenEnCurso.EnH01_Existe := TRUE;
           ELSE
               #OrdenJdT.OrdenPoscionado_NOK := TRUE;
           END_IF;

       END_IF;

       //////////////////////////////////////////////////////////////////////
       // Orden de Posicionar a la Horquilla 2
       IF (#OrdenJdT.VarMesaHorquilla = #NumMesaH2) THEN
           IF ("DB885_ConfigMaquinas".Maquina[#Maquina].Mesa[#OrdenJdT.VarMesaCargaDesCarga].Posicion_mm_H2 <> 0) THEN
               #OrdenEnCurso.EnH02_Poscicion := "DB885_ConfigMaquinas".Maquina[#Maquina].Mesa[#OrdenJdT.VarMesaCargaDesCarga].Posicion_mm_H2;
               #OrdenH02_TipoMovi.Posicionar := TRUE;
               #OrdenEnCurso.EnH02_Existe := TRUE;
           ELSE
               #OrdenJdT.OrdenPoscionado_NOK := TRUE;
           END_IF;

       END_IF;

       //////////////////////////////////////////////////////////////////////
       // Orden de Posicionar a la Horquilla No Existente
       IF (#OrdenJdT.VarMesaHorquilla <> #NumMesaH1) AND (#OrdenJdT.VarMesaHorquilla <> #NumMesaH2) THEN
           #OrdenJdT.OrdenPoscionado_NOK := TRUE;

       END_IF;

       //////////////////////////////////////////////////////////////////////
       // Orden de Posicionado Rechazada
       IF ("DB832_Maquinas".Maquinas[#NumVTD].VTD_ELEV.Respuesta = 0) AND (#OrdenJdT.OrdenPoscionado_NOK = TRUE) THEN
           "DB832_Maquinas".Maquinas[#NumVTD].VTD_ELEV.Respuesta := "Evento_VTDC_FinPosicionado_NOK";
           "DB832_Maquinas".Maquinas[#NumVTD].VTD_ELEV.Operacion := 0;
           #OrdenJdT.Operacion := 0;
           #OrdenJdT.OrdenPoscionado_NOK := FALSE;

       END_IF;

   END_IF;
END_REGION

REGION Network 16: >>>>>>>>>>>>>>>>>>>>>>>>>>>>>>>>>>>>>>>>>>>>>>>>>>>>>>>>>>>>>>>>>>>>>>>>>>>>>>>>
END_REGION

REGION Network 17 (SCL): HMI >>> Orden de Posicionar el VTD (Horquilla, Mesa Carga o DesCarga)
   /////////////////////////////////////////////////////////////////////////////
   // --- Orden de Posicionar el VTD (Horquilla, Mesa Carga o DesCarga)

   #OrdenHMI.MesaHorquilla := "DB771_HMI_VTD".Dispositivo[#Maquina].Mov_Manual.MesaHorquilla;
   #OrdenHMI.MesaDestino := "DB771_HMI_VTD".Dispositivo[#Maquina].Mov_Manual.MesaDestino;
   #OrdenHMI.VarMesaHorquilla := #OrdenHMI.MesaHorquilla - "CTE_OffsetMesa";
   #OrdenHMI.VarMesaDestino := #OrdenHMI.VarMesaDestino - "CTE_OffsetMesa";

   IF (#OrdenHMI.VarMesaHorquilla >= 1) AND (#OrdenHMI.VarMesaHorquilla <= "CTE_MaxMesas") AND
       (#OrdenHMI.VarMesaDestino >= 1) AND  (#OrdenHMI.VarMesaDestino <= "CTE_MaxMesas") AND
       (#EnMarchaVTDC = TRUE) AND
       (#OrdenEnCurso.EnH01_Existe = FALSE) AND (#OrdenEnCurso.EnH02_Existe = FALSE) THEN


       //////////////////////////////////////////////////////////////////////
       // Orden de Posicionar a la Horquilla 1
       IF (#OrdenHMI.VarMesaHorquilla = #NumMesaH1) THEN
           IF ("DB885_ConfigMaquinas".Maquina[#Maquina].Mesa[#OrdenHMI.VarMesaDestino].Posicion_mm_H1 <> 0) THEN
               #OrdenEnCurso.EnH01_Poscicion := "DB885_ConfigMaquinas".Maquina[#Maquina].Mesa[#OrdenHMI.VarMesaDestino].Posicion_mm_H1;
               #OrdenH01_TipoMovi.Posicionar := TRUE;
           END_IF;

           "DB771_HMI_VTD".Dispositivo[#Maquina].Mov_Manual.MesaHorquilla := 0;
           "DB771_HMI_VTD".Dispositivo[#Maquina].Mov_Manual.MesaDestino := 0;

       END_IF;

       //////////////////////////////////////////////////////////////////////
       // Orden de Posicionar a la Horquilla 2
       IF (#OrdenHMI.VarMesaHorquilla = #NumMesaH2) THEN
           IF ("DB885_ConfigMaquinas".Maquina[#Maquina].Mesa[#OrdenHMI.VarMesaDestino].Posicion_mm_H2 <> 0) THEN
               #OrdenEnCurso.EnH01_Poscicion := "DB885_ConfigMaquinas".Maquina[#Maquina].Mesa[#OrdenHMI.VarMesaDestino].Posicion_mm_H2;
               #OrdenH02_TipoMovi.Posicionar := TRUE;
           END_IF;

           "DB771_HMI_VTD".Dispositivo[#Maquina].Mov_Manual.MesaHorquilla := 0;
           "DB771_HMI_VTD".Dispositivo[#Maquina].Mov_Manual.MesaDestino := 0;

       END_IF;

       //////////////////////////////////////////////////////////////////////
       // Orden de Posicionar a la Horquilla No Existente
       IF (#OrdenJdT.VarMesaHorquilla <> #NumMesaH1) AND (#OrdenJdT.VarMesaHorquilla <> #NumMesaH2) THEN
           "DB771_HMI_VTD".Dispositivo[#Maquina].Mov_Manual.MesaHorquilla := 0;
           "DB771_HMI_VTD".Dispositivo[#Maquina].Mov_Manual.MesaDestino := 0;

       END_IF;


   END_IF;
END_REGION

REGION Network 18: >>>>>>>>>>>>>>>>>>>>>>>>>>>>>>>>>>>>>>>>>>>>>>>>>>>>>>>>>>>>>>>>>>>>>>>>>>>>>>>>
END_REGION

REGION Network 19: CONTROL DE ORDENES EN CURSO >>> Existe Orden En Curso En H01
   RUNG wire#powerrail
      Contact( "ON" )
      R_Coil( #OrdenEnCurso.EnH01_Existe )
   END_RUNG
   RUNG wire#powerrail
      I_Contact( #OrdenH01_TipoMovi.CargaDcha )
      I_Contact( #OrdenH01_TipoMovi.DesCargaDcha )
      I_Contact( #OrdenH01_TipoMovi.CargaIzq )
      I_Contact( #OrdenH01_TipoMovi.DesCargaIzq )
      I_Contact( #OrdenH01_TipoMovi.Posicionar )
      Not()
      S_Coil( #OrdenEnCurso.EnH01_Existe )
   END_RUNG
   RUNG wire#powerrail
      I_Contact( #OrdenEnCurso.EnH01_Existe )
      Move(in := 0.0, out1 => #OrdenEnCurso.EnH01_Poscicion)
   END_RUNG
   // the same network as SCL:
   IF "ON" THEN #OrdenEnCurso.EnH01_Existe := FALSE; END_IF;
   IF NOT (NOT #OrdenH01_TipoMovi.CargaDcha AND NOT #OrdenH01_TipoMovi.DesCargaDcha AND NOT #OrdenH01_TipoMovi.CargaIzq AND NOT #OrdenH01_TipoMovi.DesCargaIzq AND NOT #OrdenH01_TipoMovi.Posicionar) THEN
       #OrdenEnCurso.EnH01_Existe := TRUE;
   END_IF;
   IF NOT #OrdenEnCurso.EnH01_Existe THEN #OrdenEnCurso.EnH01_Poscicion := 0.0; END_IF;
END_REGION

REGION Network 20: CONTROL DE ORDENES EN CURSO >>> Existe Orden En Curso En H02
   RUNG wire#powerrail
      Contact( "ON" )
      R_Coil( #OrdenEnCurso.EnH02_Existe )
   END_RUNG
   RUNG wire#powerrail
      I_Contact( #OrdenH02_TipoMovi.CargaDcha )
      I_Contact( #OrdenH02_TipoMovi.DesCargaDcha )
      I_Contact( #OrdenH02_TipoMovi.CargaIzq )
      I_Contact( #OrdenH02_TipoMovi.DesCargaIzq )
      I_Contact( #OrdenH02_TipoMovi.Posicionar )
      Not()
      S_Coil( #OrdenEnCurso.EnH02_Existe )
   END_RUNG
   RUNG wire#powerrail
      I_Contact( #OrdenEnCurso.EnH02_Existe )
      Move(in := 0.0, out1 => #OrdenEnCurso.EnH02_Poscicion)
   END_RUNG
   // the same network as SCL:
   IF "ON" THEN #OrdenEnCurso.EnH02_Existe := FALSE; END_IF;
   IF NOT (NOT #OrdenH02_TipoMovi.CargaDcha AND NOT #OrdenH02_TipoMovi.DesCargaDcha AND NOT #OrdenH02_TipoMovi.CargaIzq AND NOT #OrdenH02_TipoMovi.DesCargaIzq AND NOT #OrdenH02_TipoMovi.Posicionar) THEN
       #OrdenEnCurso.EnH02_Existe := TRUE;
   END_IF;
   IF NOT #OrdenEnCurso.EnH02_Existe THEN #OrdenEnCurso.EnH02_Poscicion := 0.0; END_IF;
END_REGION

REGION Network 21: >>>>>>>>>>>>>>>>>>>>>>>>>>>>>>>>>>>>>>>>>>>>>>>>>>>>>>>>>>>>>>>>>>>>>>>>>>>>>>>>
END_REGION

REGION Network 22: FIN DE ORDENES >>> CARGA en la H01
   RUNG wire#powerrail
      Contact( #EstadoVI_MesaH1.Etapas_Carga_E1 )
      N_Trig( #MemoFlancos.H1.Carga_E1 )
      Move(in := 0, out1 => #OrdenEnCurso.EnH01_MesaCarga)
      R_Coil( #OrdenH01_TipoMovi.CargaDcha )
   END_RUNG
   RUNG wire#powerrail
      Contact( #EstadoVI_MesaH1.Etapas_Carga_E3 )
      N_Trig( #MemoFlancos.H1.Carga_E3 )
      Move(in := 0, out1 => #OrdenEnCurso.EnH01_MesaCarga)
      R_Coil( #OrdenH01_TipoMovi.CargaIzq )
   END_RUNG
   // the same network as SCL:
   #_w1 := NOT #EstadoVI_MesaH1.Etapas_Carga_E1 AND #MemoFlancos.H1.Carga_E1;   // falling edge
   #MemoFlancos.H1.Carga_E1 := #EstadoVI_MesaH1.Etapas_Carga_E1;
   IF #_w1 THEN
       #OrdenEnCurso.EnH01_MesaCarga := 0;
       #OrdenH01_TipoMovi.CargaDcha := FALSE;
   END_IF;
   #_w2 := NOT #EstadoVI_MesaH1.Etapas_Carga_E3 AND #MemoFlancos.H1.Carga_E3;   // falling edge
   #MemoFlancos.H1.Carga_E3 := #EstadoVI_MesaH1.Etapas_Carga_E3;
   IF #_w2 THEN
       #OrdenEnCurso.EnH01_MesaCarga := 0;
       #OrdenH01_TipoMovi.CargaIzq := FALSE;
   END_IF;
END_REGION

REGION Network 23: >>> DESCARGA de la H01
   RUNG wire#powerrail
      Contact( #EstadoVI_MesaH1.Etapas_Descarga_S1 )
      N_Trig( #MemoFlancos.H1.DesCarga_S1 )
      Move(in := 0, out1 => #OrdenEnCurso.EnH01_MesaDesCarga)
      R_Coil( #OrdenH01_TipoMovi.DesCargaDcha )
   END_RUNG
   RUNG wire#powerrail
      Contact( #EstadoVI_MesaH1.Etapas_Descarga_S3 )
      N_Trig( #MemoFlancos.H1.DesCarga_S3 )
      Move(in := 0, out1 => #OrdenEnCurso.EnH01_MesaDesCarga)
      R_Coil( #OrdenH01_TipoMovi.DesCargaIzq )
   END_RUNG
   // the same network as SCL:
   #_w1 := NOT #EstadoVI_MesaH1.Etapas_Descarga_S1 AND #MemoFlancos.H1.DesCarga_S1;   // falling edge
   #MemoFlancos.H1.DesCarga_S1 := #EstadoVI_MesaH1.Etapas_Descarga_S1;
   IF #_w1 THEN
       #OrdenEnCurso.EnH01_MesaDesCarga := 0;
       #OrdenH01_TipoMovi.DesCargaDcha := FALSE;
   END_IF;
   #_w2 := NOT #EstadoVI_MesaH1.Etapas_Descarga_S3 AND #MemoFlancos.H1.DesCarga_S3;   // falling edge
   #MemoFlancos.H1.DesCarga_S3 := #EstadoVI_MesaH1.Etapas_Descarga_S3;
   IF #_w2 THEN
       #OrdenEnCurso.EnH01_MesaDesCarga := 0;
       #OrdenH01_TipoMovi.DesCargaIzq := FALSE;
   END_IF;
END_REGION

REGION Network 24: >>> POSICIONAR la H01
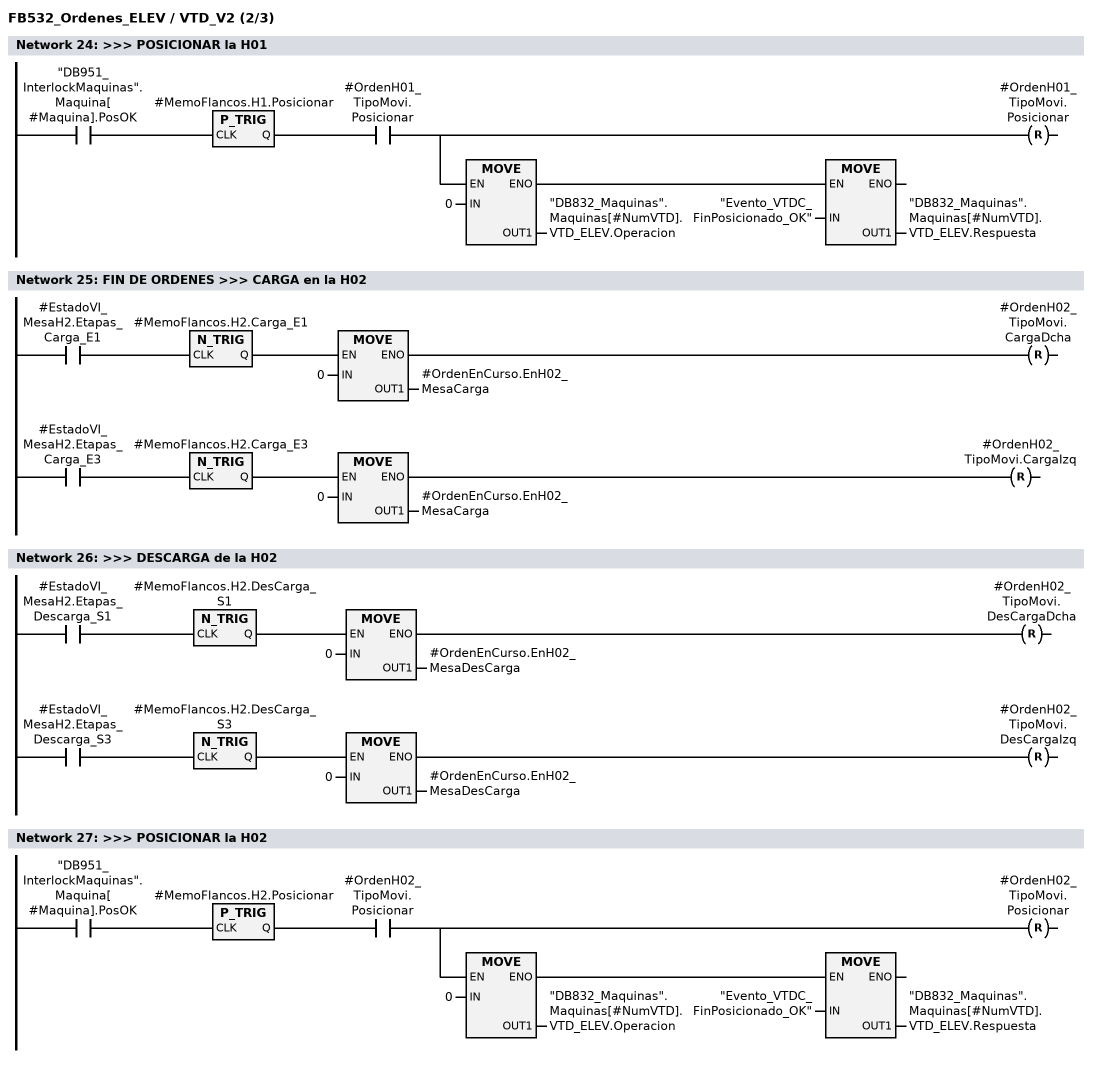
   RUNG wire#powerrail
      Contact( "DB951_InterlockMaquinas".Maquina[#Maquina].PosOK )
      P_Trig( #MemoFlancos.H1.Posicionar )
      Contact( #OrdenH01_TipoMovi.Posicionar )
      wire#w1
      R_Coil( #OrdenH01_TipoMovi.Posicionar )
   END_RUNG
   RUNG wire#w1
      Move(in := 0, out1 => "DB832_Maquinas".Maquinas[#NumVTD].VTD_ELEV.Operacion)
      Move(in := "Evento_VTDC_FinPosicionado_OK", out1 => "DB832_Maquinas".Maquinas[#NumVTD].VTD_ELEV.Respuesta)
   END_RUNG
   // the same network as SCL:
   #_w1 := "DB951_InterlockMaquinas".Maquina[#Maquina].PosOK AND NOT #MemoFlancos.H1.Posicionar;   // rising edge
   #MemoFlancos.H1.Posicionar := "DB951_InterlockMaquinas".Maquina[#Maquina].PosOK;
   #_w2 := #_w1 AND #OrdenH01_TipoMovi.Posicionar;
   IF #_w2 THEN
       #OrdenH01_TipoMovi.Posicionar := FALSE;
       "DB832_Maquinas".Maquinas[#NumVTD].VTD_ELEV.Operacion := 0;
       "DB832_Maquinas".Maquinas[#NumVTD].VTD_ELEV.Respuesta := "Evento_VTDC_FinPosicionado_OK";
   END_IF;
END_REGION

REGION Network 25: FIN DE ORDENES >>> CARGA en la H02
   RUNG wire#powerrail
      Contact( #EstadoVI_MesaH2.Etapas_Carga_E1 )
      N_Trig( #MemoFlancos.H2.Carga_E1 )
      Move(in := 0, out1 => #OrdenEnCurso.EnH02_MesaCarga)
      R_Coil( #OrdenH02_TipoMovi.CargaDcha )
   END_RUNG
   RUNG wire#powerrail
      Contact( #EstadoVI_MesaH2.Etapas_Carga_E3 )
      N_Trig( #MemoFlancos.H2.Carga_E3 )
      Move(in := 0, out1 => #OrdenEnCurso.EnH02_MesaCarga)
      R_Coil( #OrdenH02_TipoMovi.CargaIzq )
   END_RUNG
   // the same network as SCL:
   #_w1 := NOT #EstadoVI_MesaH2.Etapas_Carga_E1 AND #MemoFlancos.H2.Carga_E1;   // falling edge
   #MemoFlancos.H2.Carga_E1 := #EstadoVI_MesaH2.Etapas_Carga_E1;
   IF #_w1 THEN
       #OrdenEnCurso.EnH02_MesaCarga := 0;
       #OrdenH02_TipoMovi.CargaDcha := FALSE;
   END_IF;
   #_w2 := NOT #EstadoVI_MesaH2.Etapas_Carga_E3 AND #MemoFlancos.H2.Carga_E3;   // falling edge
   #MemoFlancos.H2.Carga_E3 := #EstadoVI_MesaH2.Etapas_Carga_E3;
   IF #_w2 THEN
       #OrdenEnCurso.EnH02_MesaCarga := 0;
       #OrdenH02_TipoMovi.CargaIzq := FALSE;
   END_IF;
END_REGION

REGION Network 26: >>> DESCARGA de la H02
   RUNG wire#powerrail
      Contact( #EstadoVI_MesaH2.Etapas_Descarga_S1 )
      N_Trig( #MemoFlancos.H2.DesCarga_S1 )
      Move(in := 0, out1 => #OrdenEnCurso.EnH02_MesaDesCarga)
      R_Coil( #OrdenH02_TipoMovi.DesCargaDcha )
   END_RUNG
   RUNG wire#powerrail
      Contact( #EstadoVI_MesaH2.Etapas_Descarga_S3 )
      N_Trig( #MemoFlancos.H2.DesCarga_S3 )
      Move(in := 0, out1 => #OrdenEnCurso.EnH02_MesaDesCarga)
      R_Coil( #OrdenH02_TipoMovi.DesCargaIzq )
   END_RUNG
   // the same network as SCL:
   #_w1 := NOT #EstadoVI_MesaH2.Etapas_Descarga_S1 AND #MemoFlancos.H2.DesCarga_S1;   // falling edge
   #MemoFlancos.H2.DesCarga_S1 := #EstadoVI_MesaH2.Etapas_Descarga_S1;
   IF #_w1 THEN
       #OrdenEnCurso.EnH02_MesaDesCarga := 0;
       #OrdenH02_TipoMovi.DesCargaDcha := FALSE;
   END_IF;
   #_w2 := NOT #EstadoVI_MesaH2.Etapas_Descarga_S3 AND #MemoFlancos.H2.DesCarga_S3;   // falling edge
   #MemoFlancos.H2.DesCarga_S3 := #EstadoVI_MesaH2.Etapas_Descarga_S3;
   IF #_w2 THEN
       #OrdenEnCurso.EnH02_MesaDesCarga := 0;
       #OrdenH02_TipoMovi.DesCargaIzq := FALSE;
   END_IF;
END_REGION

REGION Network 27: >>> POSICIONAR la H02
   RUNG wire#powerrail
      Contact( "DB951_InterlockMaquinas".Maquina[#Maquina].PosOK )
      P_Trig( #MemoFlancos.H2.Posicionar )
      Contact( #OrdenH02_TipoMovi.Posicionar )
      wire#w1
      R_Coil( #OrdenH02_TipoMovi.Posicionar )
   END_RUNG
   RUNG wire#w1
      Move(in := 0, out1 => "DB832_Maquinas".Maquinas[#NumVTD].VTD_ELEV.Operacion)
      Move(in := "Evento_VTDC_FinPosicionado_OK", out1 => "DB832_Maquinas".Maquinas[#NumVTD].VTD_ELEV.Respuesta)
   END_RUNG
   // the same network as SCL:
   #_w1 := "DB951_InterlockMaquinas".Maquina[#Maquina].PosOK AND NOT #MemoFlancos.H2.Posicionar;   // rising edge
   #MemoFlancos.H2.Posicionar := "DB951_InterlockMaquinas".Maquina[#Maquina].PosOK;
   #_w2 := #_w1 AND #OrdenH02_TipoMovi.Posicionar;
   IF #_w2 THEN
       #OrdenH02_TipoMovi.Posicionar := FALSE;
       "DB832_Maquinas".Maquinas[#NumVTD].VTD_ELEV.Operacion := 0;
       "DB832_Maquinas".Maquinas[#NumVTD].VTD_ELEV.Respuesta := "Evento_VTDC_FinPosicionado_OK";
   END_IF;
END_REGION

REGION Network 28: >>>>>>>>>>>>>>>>>>>>>>>>>>>>>>>>>>>>>>>>>>>>>>>>>>>>>>>>>>>>>>>>>>>>>>>>>>>>>>>>
END_REGION

REGION Network 29 (SCL): INTERLOCK >>> Inicializar la Mesas de la Horquillas
   /////////////////////////////////////////////////////////////////////////////
   // --- INTERLOCK >>> Inicializar la Mesas de las Horquillas
   // 
   #ValorReturn := FILL(BVAL := #Cero, BLK => "DB951_InterlockMaquinas".Maquina[#Maquina].H1.In);
   #ValorReturn := FILL(BVAL := #Cero, BLK => "DB951_InterlockMaquinas".Maquina[#Maquina].H2.In);

   "DB951_InterlockMaquinas".Maquina[#Maquina].H1.Mesa_EntradaDerecha := 0;
   "DB951_InterlockMaquinas".Maquina[#Maquina].H1.Mesa_EntradaIzquierda := 0;
   "DB951_InterlockMaquinas".Maquina[#Maquina].H2.Mesa_EntradaDerecha := 0;
   "DB951_InterlockMaquinas".Maquina[#Maquina].H2.Mesa_EntradaIzquierda := 0;
END_REGION

REGION Network 30 (SCL): INTERLOCK >>> Inicializar la Mesas de Carga o DesCarga
   /////////////////////////////////////////////////////////////////////////////
   // --- INTERLOCK >>> Inicializar la Mesas de Carga o DesCarga
   // 

   FOR #VarInterlock.Indice := 1 TO "CTE_MaxMesas" DO
       #ValorReturn := FILL(BVAL := #Cero, BLK => "DB951_InterlockMaquinas".Maquina[#Maquina].Mesa[#VarInterlock.Indice].In);
       "DB951_InterlockMaquinas".Maquina[#Maquina].Mesa[#VarInterlock.Indice].PosOK_H1 := FALSE;
       "DB951_InterlockMaquinas".Maquina[#Maquina].Mesa[#VarInterlock.Indice].PosOK_H2 := FALSE;

   END_FOR;
END_REGION

REGION Network 31 (SCL): INTERLOCK >>> Intercambio de Entradas y Salidas En Horquilla 1
   /////////////////////////////////////////////////////////////////////////////
   // --- INTERLOCK >>> Intercambio de Entradas y Salidas
   // 

   /////////////////////////////////////////////////////////////////////////////
   // Ciertas señales Hay que mantener siempre
   // ORDENES DE CARGA
   IF (#OrdenH01_TipoMovi.CargaDcha) AND (#OrdenEnCurso.EnH01_MesaCarga <> 0) THEN
       "DB951_InterlockMaquinas".Maquina[#Maquina].H1.Mesa_EntradaDerecha := #OrdenEnCurso.EnH01_MesaCarga;
       "DB951_InterlockMaquinas".Maquina[#Maquina].H1.In.DesCargaAct_Dcha := "DB900_Estado_Mesas".EstadoVI[#OrdenEnCurso.EnH01_MesaCarga].Descarga_Act;
       "DB951_InterlockMaquinas".Maquina[#Maquina].Mesa[#OrdenEnCurso.EnH01_MesaCarga].In.CargaAct := "DB900_Estado_Mesas".EstadoVI[#NumMesaH1].Etapas_Carga_E1;

   END_IF;

   IF (#OrdenH01_TipoMovi.CargaIzq) AND (#OrdenEnCurso.EnH01_MesaCarga <> 0) THEN
       "DB951_InterlockMaquinas".Maquina[#Maquina].H1.Mesa_EntradaIzquierda := #OrdenEnCurso.EnH01_MesaCarga;
       "DB951_InterlockMaquinas".Maquina[#Maquina].H1.In.DesCargaAct_Izq := "DB900_Estado_Mesas".EstadoVI[#OrdenEnCurso.EnH01_MesaCarga].Descarga_Act;
       "DB951_InterlockMaquinas".Maquina[#Maquina].Mesa[#OrdenEnCurso.EnH01_MesaCarga].In.CargaAct := "DB900_Estado_Mesas".EstadoVI[#NumMesaH1].Etapas_Carga_E3;

   END_IF;

   // ORDENES DE DESCARGA
   IF (#OrdenH01_TipoMovi.DesCargaDcha) AND (#OrdenEnCurso.EnH01_MesaDesCarga <> 0) THEN
       "DB951_InterlockMaquinas".Maquina[#Maquina].Mesa[#OrdenEnCurso.EnH01_MesaDesCarga].MesaEntrada := #NumMesaH1;
       "DB951_InterlockMaquinas".Maquina[#Maquina].Mesa[#OrdenEnCurso.EnH01_MesaDesCarga].In.DesCargaAct := "DB900_Estado_Mesas".EstadoVI[#NumMesaH1].Descarga_Act;
       "DB951_InterlockMaquinas".Maquina[#Maquina].H1.In.CargaAct_Dcha := "DB900_Estado_Mesas".EstadoVI[#OrdenEnCurso.EnH01_MesaDesCarga].Etapas_Carga_E1 OR
                                                                          "DB900_Estado_Mesas".EstadoVI[#OrdenEnCurso.EnH01_MesaDesCarga].Etapas_Carga_E2 OR
                                                                          "DB900_Estado_Mesas".EstadoVI[#OrdenEnCurso.EnH01_MesaDesCarga].Etapas_Carga_E3 OR
                                                                          "DB900_Estado_Mesas".EstadoVI[#OrdenEnCurso.EnH01_MesaDesCarga].Etapas_Carga_E4;
   END_IF;

   IF (#OrdenH01_TipoMovi.DesCargaIzq) AND (#OrdenEnCurso.EnH01_MesaDesCarga <> 0) THEN
       "DB951_InterlockMaquinas".Maquina[#Maquina].Mesa[#OrdenEnCurso.EnH01_MesaDesCarga].MesaEntrada := #NumMesaH1;
       "DB951_InterlockMaquinas".Maquina[#Maquina].Mesa[#OrdenEnCurso.EnH01_MesaDesCarga].In.DesCargaAct := "DB900_Estado_Mesas".EstadoVI[#NumMesaH1].Descarga_Act;
       "DB951_InterlockMaquinas".Maquina[#Maquina].H1.In.CargaAct_Izq := "DB900_Estado_Mesas".EstadoVI[#OrdenEnCurso.EnH01_MesaDesCarga].Etapas_Carga_E1 OR
                                                                         "DB900_Estado_Mesas".EstadoVI[#OrdenEnCurso.EnH01_MesaDesCarga].Etapas_Carga_E2 OR
                                                                         "DB900_Estado_Mesas".EstadoVI[#OrdenEnCurso.EnH01_MesaDesCarga].Etapas_Carga_E3 OR
                                                                         "DB900_Estado_Mesas".EstadoVI[#OrdenEnCurso.EnH01_MesaDesCarga].Etapas_Carga_E4;
   END_IF;


   /////////////////////////////////////////////////////////////////////////////
   // Funcionamiento Normal
   IF "DB951_InterlockMaquinas".Maquina[#Maquina].PosOK THEN

       ////////////////////////////////////////////////////////////////////////
       ////////////////////////////////////////////////////////////////////////
       // --- Orden De Carga en Curso En Horquilla 1
       IF (#OrdenH01_TipoMovi.CargaDcha = TRUE) OR (#OrdenH01_TipoMovi.CargaIzq = TRUE) THEN
           #VarInterlock.Posicion := "DB885_ConfigMaquinas".Maquina[#Maquina].Mesa[#OrdenEnCurso.EnH01_MesaCarga].Posicion_mm_H1;

           // >>> Verificar que este posicionado
           IF (#VarInterlock.Posicion = #Peticion.Posicion) THEN
               "DB951_InterlockMaquinas".Maquina[#Maquina].Mesa[#OrdenEnCurso.EnH01_MesaCarga].PosOK_H1 := "DB951_InterlockMaquinas".Maquina[#Maquina].PosOK;

               // >>>> Orden de Carga por la Derecha
               IF (#OrdenH01_TipoMovi.CargaDcha) THEN
                   "DB951_InterlockMaquinas".Maquina[#Maquina].H1.Mesa_EntradaDerecha := #OrdenEnCurso.EnH01_MesaCarga;

                   // >>> Entradas a la Horquila
                   "DB951_InterlockMaquinas".Maquina[#Maquina].H1.In.AVTF_Dcha := "DB951_InterlockMaquinas".Maquina[#Maquina].Mesa[#OrdenEnCurso.EnH01_MesaCarga].Out.AVTF;
                   "DB951_InterlockMaquinas".Maquina[#Maquina].H1.In.P_Mens_Dcha := "DB951_InterlockMaquinas".Maquina[#Maquina].Mesa[#OrdenEnCurso.EnH01_MesaCarga].Out.P_Mens;
                   "DB951_InterlockMaquinas".Maquina[#Maquina].H1.In.DesCargaAct_Dcha := "DB900_Estado_Mesas".EstadoVI[#OrdenEnCurso.EnH01_MesaCarga].Descarga_Act;
                   // >>> Salidas de la Horquilla
                   "DB951_InterlockMaquinas".Maquina[#Maquina].Mesa[#OrdenEnCurso.EnH01_MesaCarga].In.PTF := "DB951_InterlockMaquinas".Maquina[#Maquina].H1.Out.PTF_Dcha;
                   "DB951_InterlockMaquinas".Maquina[#Maquina].Mesa[#OrdenEnCurso.EnH01_MesaCarga].In.FTF := "DB951_InterlockMaquinas".Maquina[#Maquina].H1.Out.FTF_Dcha;
                   "DB951_InterlockMaquinas".Maquina[#Maquina].Mesa[#OrdenEnCurso.EnH01_MesaCarga].In.CargaAct := "DB900_Estado_Mesas".EstadoVI[#NumMesaH1].Etapas_Carga_E1;

               END_IF;

               // >>>> Orden de Carga por la Izquierda
               IF (#OrdenH01_TipoMovi.CargaIzq) THEN
                   "DB951_InterlockMaquinas".Maquina[#Maquina].H1.Mesa_EntradaIzquierda := #OrdenEnCurso.EnH01_MesaCarga;

                   // >>> Entradas a la Horquila
                   "DB951_InterlockMaquinas".Maquina[#Maquina].H1.In.AVTF_Izq := "DB951_InterlockMaquinas".Maquina[#Maquina].Mesa[#OrdenEnCurso.EnH01_MesaCarga].Out.AVTF;
                   "DB951_InterlockMaquinas".Maquina[#Maquina].H1.In.P_Mens_Izq := "DB951_InterlockMaquinas".Maquina[#Maquina].Mesa[#OrdenEnCurso.EnH01_MesaCarga].Out.P_Mens;
                   "DB951_InterlockMaquinas".Maquina[#Maquina].H1.In.DesCargaAct_Izq := "DB900_Estado_Mesas".EstadoVI[#OrdenEnCurso.EnH01_MesaCarga].Descarga_Act;
                   // >>> Salidas de la Horquilla
                   "DB951_InterlockMaquinas".Maquina[#Maquina].Mesa[#OrdenEnCurso.EnH01_MesaCarga].In.PTF := "DB951_InterlockMaquinas".Maquina[#Maquina].H1.Out.PTF_Izq;
                   "DB951_InterlockMaquinas".Maquina[#Maquina].Mesa[#OrdenEnCurso.EnH01_MesaCarga].In.FTF := "DB951_InterlockMaquinas".Maquina[#Maquina].H1.Out.FTF_Izq;
                   "DB951_InterlockMaquinas".Maquina[#Maquina].Mesa[#OrdenEnCurso.EnH01_MesaCarga].In.CargaAct := "DB900_Estado_Mesas".EstadoVI[#NumMesaH1].Etapas_Carga_E3;

               END_IF;

           END_IF;
       END_IF;


       ////////////////////////////////////////////////////////////////////////
       ////////////////////////////////////////////////////////////////////////
       // --- Orden De DesCarga en Curso En Horquilla 1
       IF (#OrdenH01_TipoMovi.DesCargaDcha = TRUE) OR (#OrdenH01_TipoMovi.DesCargaIzq = TRUE) THEN
           #VarInterlock.Posicion := "DB885_ConfigMaquinas".Maquina[#Maquina].Mesa[#OrdenEnCurso.EnH01_MesaDesCarga].Posicion_mm_H1;

           // >>> Verificar que este posicionado
           IF (#VarInterlock.Posicion = #Peticion.Posicion) THEN
               "DB951_InterlockMaquinas".Maquina[#Maquina].Mesa[#OrdenEnCurso.EnH01_MesaDesCarga].PosOK_H1 := "DB951_InterlockMaquinas".Maquina[#Maquina].PosOK;

               // >>>> Orden de DesCarga por la Derecha
               IF (#OrdenH01_TipoMovi.DesCargaDcha) THEN
                   "DB951_InterlockMaquinas".Maquina[#Maquina].Mesa[#OrdenEnCurso.EnH01_MesaDesCarga].MesaEntrada := #NumMesaH1;

                   // >>> Entradas a la Horquila
                   "DB951_InterlockMaquinas".Maquina[#Maquina].Mesa[#OrdenEnCurso.EnH01_MesaDesCarga].In.AVTF := "DB951_InterlockMaquinas".Maquina[#Maquina].H1.Out.AVTF_Dcha;
                   "DB951_InterlockMaquinas".Maquina[#Maquina].Mesa[#OrdenEnCurso.EnH01_MesaDesCarga].In.P_Mens := "DB951_InterlockMaquinas".Maquina[#Maquina].H1.Out.P_Mens_Dcha;
                   "DB951_InterlockMaquinas".Maquina[#Maquina].Mesa[#OrdenEnCurso.EnH01_MesaDesCarga].In.DesCargaAct := "DB900_Estado_Mesas".EstadoVI[#NumMesaH1].Descarga_Act;
                   // >>> Salidas de la Horquilla
                   "DB951_InterlockMaquinas".Maquina[#Maquina].H1.In.PTF_Dcha := "DB951_InterlockMaquinas".Maquina[#Maquina].Mesa[#OrdenEnCurso.EnH01_MesaDesCarga].Out.PTF;
                   "DB951_InterlockMaquinas".Maquina[#Maquina].H1.In.FTF_Dcha := "DB951_InterlockMaquinas".Maquina[#Maquina].Mesa[#OrdenEnCurso.EnH01_MesaDesCarga].Out.FTF;
                   "DB951_InterlockMaquinas".Maquina[#Maquina].H1.In.CargaAct_Dcha := "DB900_Estado_Mesas".EstadoVI[#OrdenEnCurso.EnH01_MesaDesCarga].Etapas_Carga_E1 OR
                                                                                   "DB900_Estado_Mesas".EstadoVI[#OrdenEnCurso.EnH01_MesaDesCarga].Etapas_Carga_E2 OR
                                                                                   "DB900_Estado_Mesas".EstadoVI[#OrdenEnCurso.EnH01_MesaDesCarga].Etapas_Carga_E3 OR
                                                                                   "DB900_Estado_Mesas".EstadoVI[#OrdenEnCurso.EnH01_MesaDesCarga].Etapas_Carga_E4;
               END_IF;


               // >>>> Orden de DesCarga por la Izquierda
               IF (#OrdenH01_TipoMovi.DesCargaIzq) THEN
                   "DB951_InterlockMaquinas".Maquina[#Maquina].Mesa[#OrdenEnCurso.EnH01_MesaDesCarga].MesaEntrada := #NumMesaH1;

                   // >>> Entradas a la Horquila
                   "DB951_InterlockMaquinas".Maquina[#Maquina].Mesa[#OrdenEnCurso.EnH01_MesaDesCarga].In.AVTF := "DB951_InterlockMaquinas".Maquina[#Maquina].H1.Out.AVTF_Izq;
                   "DB951_InterlockMaquinas".Maquina[#Maquina].Mesa[#OrdenEnCurso.EnH01_MesaDesCarga].In.P_Mens := "DB951_InterlockMaquinas".Maquina[#Maquina].H1.Out.P_Mens_Izq;
                   "DB951_InterlockMaquinas".Maquina[#Maquina].Mesa[#OrdenEnCurso.EnH01_MesaDesCarga].In.DesCargaAct := "DB900_Estado_Mesas".EstadoVI[#NumMesaH1].Descarga_Act;
                   // >>> Salidas de la Horquilla
                   "DB951_InterlockMaquinas".Maquina[#Maquina].H1.In.PTF_Izq := "DB951_InterlockMaquinas".Maquina[#Maquina].Mesa[#OrdenEnCurso.EnH01_MesaDesCarga].Out.PTF;
                   "DB951_InterlockMaquinas".Maquina[#Maquina].H1.In.FTF_Izq := "DB951_InterlockMaquinas".Maquina[#Maquina].Mesa[#OrdenEnCurso.EnH01_MesaDesCarga].Out.FTF;
                   "DB951_InterlockMaquinas".Maquina[#Maquina].H1.In.CargaAct_Izq := "DB900_Estado_Mesas".EstadoVI[#OrdenEnCurso.EnH01_MesaDesCarga].Etapas_Carga_E1 OR
                   "DB900_Estado_Mesas".EstadoVI[#OrdenEnCurso.EnH01_MesaDesCarga].Etapas_Carga_E2 OR
                   "DB900_Estado_Mesas".EstadoVI[#OrdenEnCurso.EnH01_MesaDesCarga].Etapas_Carga_E3 OR
                   "DB900_Estado_Mesas".EstadoVI[#OrdenEnCurso.EnH01_MesaDesCarga].Etapas_Carga_E4;
               END_IF;

           END_IF;
       END_IF;




   END_IF;
END_REGION

REGION Network 32 (SCL): INTERLOCK >>> Intercambio de Entradas y Salidas En Horquilla 2
   /////////////////////////////////////////////////////////////////////////////
   // --- INTERLOCK >>> Intercambio de Entradas y Salidas
   // 

   /////////////////////////////////////////////////////////////////////////////
   // Ciertas señales Hay que mantener siempre
   // ORDENES DE CARGA
   IF (#OrdenH02_TipoMovi.CargaDcha) AND (#OrdenEnCurso.EnH02_MesaCarga <> 0) THEN
       "DB951_InterlockMaquinas".Maquina[#Maquina].H2.Mesa_EntradaDerecha := #OrdenEnCurso.EnH02_MesaCarga;
       "DB951_InterlockMaquinas".Maquina[#Maquina].H2.In.DesCargaAct_Dcha := "DB900_Estado_Mesas".EstadoVI[#OrdenEnCurso.EnH02_MesaCarga].Descarga_Act;
       "DB951_InterlockMaquinas".Maquina[#Maquina].Mesa[#OrdenEnCurso.EnH02_MesaCarga].In.CargaAct := "DB900_Estado_Mesas".EstadoVI[#NumMesaH2].Etapas_Carga_E1;

   END_IF;

   IF (#OrdenH02_TipoMovi.CargaIzq) AND (#OrdenEnCurso.EnH02_MesaCarga <> 0) THEN
       "DB951_InterlockMaquinas".Maquina[#Maquina].H2.Mesa_EntradaIzquierda := #OrdenEnCurso.EnH02_MesaCarga;
       "DB951_InterlockMaquinas".Maquina[#Maquina].H2.In.DesCargaAct_Izq := "DB900_Estado_Mesas".EstadoVI[#OrdenEnCurso.EnH02_MesaCarga].Descarga_Act;
       "DB951_InterlockMaquinas".Maquina[#Maquina].Mesa[#OrdenEnCurso.EnH02_MesaCarga].In.CargaAct := "DB900_Estado_Mesas".EstadoVI[#NumMesaH2].Etapas_Carga_E3;

   END_IF;

   // ORDENES DE DESCARGA
   IF (#OrdenH02_TipoMovi.DesCargaDcha) AND (#OrdenEnCurso.EnH02_MesaDesCarga <> 0) THEN
       "DB951_InterlockMaquinas".Maquina[#Maquina].Mesa[#OrdenEnCurso.EnH02_MesaDesCarga].MesaEntrada := #NumMesaH1;
       "DB951_InterlockMaquinas".Maquina[#Maquina].Mesa[#OrdenEnCurso.EnH02_MesaDesCarga].In.DesCargaAct := "DB900_Estado_Mesas".EstadoVI[#NumMesaH2].Descarga_Act;
       "DB951_InterlockMaquinas".Maquina[#Maquina].H2.In.CargaAct_Dcha := "DB900_Estado_Mesas".EstadoVI[#OrdenEnCurso.EnH02_MesaDesCarga].Etapas_Carga_E1 OR
       "DB900_Estado_Mesas".EstadoVI[#OrdenEnCurso.EnH02_MesaDesCarga].Etapas_Carga_E2 OR
       "DB900_Estado_Mesas".EstadoVI[#OrdenEnCurso.EnH02_MesaDesCarga].Etapas_Carga_E3 OR
       "DB900_Estado_Mesas".EstadoVI[#OrdenEnCurso.EnH02_MesaDesCarga].Etapas_Carga_E4;
   END_IF;

   IF (#OrdenH02_TipoMovi.DesCargaIzq) AND (#OrdenEnCurso.EnH02_MesaDesCarga <> 0) THEN
       "DB951_InterlockMaquinas".Maquina[#Maquina].Mesa[#OrdenEnCurso.EnH02_MesaDesCarga].MesaEntrada := #NumMesaH1;
       "DB951_InterlockMaquinas".Maquina[#Maquina].Mesa[#OrdenEnCurso.EnH02_MesaDesCarga].In.DesCargaAct := "DB900_Estado_Mesas".EstadoVI[#NumMesaH2].Descarga_Act;
       "DB951_InterlockMaquinas".Maquina[#Maquina].H2.In.CargaAct_Izq := "DB900_Estado_Mesas".EstadoVI[#OrdenEnCurso.EnH02_MesaDesCarga].Etapas_Carga_E1 OR
       "DB900_Estado_Mesas".EstadoVI[#OrdenEnCurso.EnH02_MesaDesCarga].Etapas_Carga_E2 OR
       "DB900_Estado_Mesas".EstadoVI[#OrdenEnCurso.EnH02_MesaDesCarga].Etapas_Carga_E3 OR
       "DB900_Estado_Mesas".EstadoVI[#OrdenEnCurso.EnH02_MesaDesCarga].Etapas_Carga_E4;
   END_IF;


   /////////////////////////////////////////////////////////////////////////////
   // Funcionamiento Normal
   IF "DB951_InterlockMaquinas".Maquina[#Maquina].PosOK THEN



       ////////////////////////////////////////////////////////////////////////
       ////////////////////////////////////////////////////////////////////////
       // --- Orden De Carga en Curso En Horquilla 2
       IF (#OrdenH02_TipoMovi.CargaDcha = TRUE) OR (#OrdenH02_TipoMovi.CargaIzq = TRUE) THEN
           #VarInterlock.Posicion := "DB885_ConfigMaquinas".Maquina[#Maquina].Mesa[#OrdenEnCurso.EnH02_MesaCarga].Posicion_mm_H2;

           // >>> Verificar que este posicionado
           IF (#VarInterlock.Posicion = #Peticion.Posicion) THEN
               "DB951_InterlockMaquinas".Maquina[#Maquina].Mesa[#OrdenEnCurso.EnH02_MesaCarga].PosOK_H2 := "DB951_InterlockMaquinas".Maquina[#Maquina].PosOK;


               // >>>> Orden de Carga por la Derecha
               IF (#OrdenH02_TipoMovi.CargaDcha) THEN
                   "DB951_InterlockMaquinas".Maquina[#Maquina].H2.Mesa_EntradaDerecha := #OrdenEnCurso.EnH02_MesaCarga;

                   // >>> Entradas a la Horquila
                   "DB951_InterlockMaquinas".Maquina[#Maquina].H2.In.AVTF_Dcha := "DB951_InterlockMaquinas".Maquina[#Maquina].Mesa[#OrdenEnCurso.EnH02_MesaCarga].Out.AVTF;
                   "DB951_InterlockMaquinas".Maquina[#Maquina].H2.In.P_Mens_Dcha := "DB951_InterlockMaquinas".Maquina[#Maquina].Mesa[#OrdenEnCurso.EnH02_MesaCarga].Out.P_Mens;
                   "DB951_InterlockMaquinas".Maquina[#Maquina].H2.In.DesCargaAct_Dcha := "DB900_Estado_Mesas".EstadoVI[#OrdenEnCurso.EnH02_MesaCarga].Descarga_Act;
                   // >>> Salidas de la Horquilla
                   "DB951_InterlockMaquinas".Maquina[#Maquina].Mesa[#OrdenEnCurso.EnH02_MesaCarga].In.PTF := "DB951_InterlockMaquinas".Maquina[#Maquina].H2.Out.PTF_Dcha;
                   "DB951_InterlockMaquinas".Maquina[#Maquina].Mesa[#OrdenEnCurso.EnH02_MesaCarga].In.FTF := "DB951_InterlockMaquinas".Maquina[#Maquina].H2.Out.FTF_Dcha;
                   "DB951_InterlockMaquinas".Maquina[#Maquina].Mesa[#OrdenEnCurso.EnH02_MesaCarga].In.CargaAct := "DB900_Estado_Mesas".EstadoVI[#NumMesaH2].Etapas_Carga_E1;

               END_IF;

               // >>>> Orden de Carga por la Izquierda
               IF (#OrdenH02_TipoMovi.CargaIzq) THEN
                   "DB951_InterlockMaquinas".Maquina[#Maquina].H2.Mesa_EntradaIzquierda := #OrdenEnCurso.EnH02_MesaCarga;

                   // >>> Entradas a la Horquila
                   "DB951_InterlockMaquinas".Maquina[#Maquina].H2.In.AVTF_Izq := "DB951_InterlockMaquinas".Maquina[#Maquina].Mesa[#OrdenEnCurso.EnH02_MesaCarga].Out.AVTF;
                   "DB951_InterlockMaquinas".Maquina[#Maquina].H2.In.P_Mens_Izq := "DB951_InterlockMaquinas".Maquina[#Maquina].Mesa[#OrdenEnCurso.EnH02_MesaCarga].Out.P_Mens;
                   "DB951_InterlockMaquinas".Maquina[#Maquina].H2.In.DesCargaAct_Izq := "DB900_Estado_Mesas".EstadoVI[#OrdenEnCurso.EnH02_MesaCarga].Descarga_Act;
                   // >>> Salidas de la Horquilla
                   "DB951_InterlockMaquinas".Maquina[#Maquina].Mesa[#OrdenEnCurso.EnH02_MesaCarga].In.PTF := "DB951_InterlockMaquinas".Maquina[#Maquina].H2.Out.PTF_Izq;
                   "DB951_InterlockMaquinas".Maquina[#Maquina].Mesa[#OrdenEnCurso.EnH02_MesaCarga].In.FTF := "DB951_InterlockMaquinas".Maquina[#Maquina].H2.Out.FTF_Izq;
                   "DB951_InterlockMaquinas".Maquina[#Maquina].Mesa[#OrdenEnCurso.EnH02_MesaCarga].In.CargaAct := "DB900_Estado_Mesas".EstadoVI[#NumMesaH2].Etapas_Carga_E3;

               END_IF;

           END_IF;
       END_IF;



       ////////////////////////////////////////////////////////////////////////
       ////////////////////////////////////////////////////////////////////////
       // --- Orden De DesCarga en Curso En Horquilla 2
       // 
       IF (#OrdenH02_TipoMovi.DesCargaDcha = TRUE) OR (#OrdenH02_TipoMovi.DesCargaIzq = TRUE) THEN
           #VarInterlock.Posicion := "DB885_ConfigMaquinas".Maquina[#Maquina].Mesa[#OrdenEnCurso.EnH02_MesaDesCarga].Posicion_mm_H2;

           // >>> Verificar que este posicionado
           IF (#VarInterlock.Posicion = #Peticion.Posicion) THEN
               "DB951_InterlockMaquinas".Maquina[#Maquina].Mesa[#OrdenEnCurso.EnH02_MesaDesCarga].PosOK_H2 := "DB951_InterlockMaquinas".Maquina[#Maquina].PosOK;

               // >>>> Orden de DesCarga por la Derecha
               IF (#OrdenH02_TipoMovi.DesCargaDcha) THEN
                   "DB951_InterlockMaquinas".Maquina[#Maquina].Mesa[#OrdenEnCurso.EnH02_MesaDesCarga].MesaEntrada := #NumMesaH2;

                   // >>> Entradas a la Horquila
                   "DB951_InterlockMaquinas".Maquina[#Maquina].Mesa[#OrdenEnCurso.EnH02_MesaDesCarga].In.AVTF := "DB951_InterlockMaquinas".Maquina[#Maquina].H2.Out.AVTF_Dcha;
                   "DB951_InterlockMaquinas".Maquina[#Maquina].Mesa[#OrdenEnCurso.EnH02_MesaDesCarga].In.P_Mens := "DB951_InterlockMaquinas".Maquina[#Maquina].H2.Out.P_Mens_Dcha;
                   "DB951_InterlockMaquinas".Maquina[#Maquina].Mesa[#OrdenEnCurso.EnH02_MesaDesCarga].In.DesCargaAct := "DB900_Estado_Mesas".EstadoVI[#NumMesaH2].Descarga_Act;
                   // >>> Salidas de la Horquilla
                   "DB951_InterlockMaquinas".Maquina[#Maquina].H2.In.PTF_Dcha := "DB951_InterlockMaquinas".Maquina[#Maquina].Mesa[#OrdenEnCurso.EnH02_MesaDesCarga].Out.PTF;
                   "DB951_InterlockMaquinas".Maquina[#Maquina].H2.In.FTF_Dcha := "DB951_InterlockMaquinas".Maquina[#Maquina].Mesa[#OrdenEnCurso.EnH02_MesaDesCarga].Out.FTF;
                   "DB951_InterlockMaquinas".Maquina[#Maquina].H2.In.CargaAct_Dcha := "DB900_Estado_Mesas".EstadoVI[#OrdenEnCurso.EnH02_MesaDesCarga].Etapas_Carga_E1 OR
                   "DB900_Estado_Mesas".EstadoVI[#OrdenEnCurso.EnH02_MesaDesCarga].Etapas_Carga_E2 OR
                   "DB900_Estado_Mesas".EstadoVI[#OrdenEnCurso.EnH02_MesaDesCarga].Etapas_Carga_E3 OR
                   "DB900_Estado_Mesas".EstadoVI[#OrdenEnCurso.EnH02_MesaDesCarga].Etapas_Carga_E4;
               END_IF;


               // >>>> Orden de DesCarga por la Izquierda
               IF (#OrdenH02_TipoMovi.DesCargaIzq) THEN
                   "DB951_InterlockMaquinas".Maquina[#Maquina].Mesa[#OrdenEnCurso.EnH02_MesaDesCarga].MesaEntrada := #NumMesaH2;

                   // >>> Entradas a la Horquila
                   "DB951_InterlockMaquinas".Maquina[#Maquina].Mesa[#OrdenEnCurso.EnH02_MesaDesCarga].In.AVTF := "DB951_InterlockMaquinas".Maquina[#Maquina].H2.Out.AVTF_Izq;
                   "DB951_InterlockMaquinas".Maquina[#Maquina].Mesa[#OrdenEnCurso.EnH02_MesaDesCarga].In.P_Mens := "DB951_InterlockMaquinas".Maquina[#Maquina].H2.Out.P_Mens_Izq;
                   "DB951_InterlockMaquinas".Maquina[#Maquina].Mesa[#OrdenEnCurso.EnH02_MesaDesCarga].In.DesCargaAct := "DB900_Estado_Mesas".EstadoVI[#NumMesaH2].Descarga_Act;
                   // >>> Salidas de la Horquilla
                   "DB951_InterlockMaquinas".Maquina[#Maquina].H2.In.PTF_Izq := "DB951_InterlockMaquinas".Maquina[#Maquina].Mesa[#OrdenEnCurso.EnH02_MesaDesCarga].Out.PTF;
                   "DB951_InterlockMaquinas".Maquina[#Maquina].H2.In.FTF_Izq := "DB951_InterlockMaquinas".Maquina[#Maquina].Mesa[#OrdenEnCurso.EnH02_MesaDesCarga].Out.FTF;
                   "DB951_InterlockMaquinas".Maquina[#Maquina].H2.In.CargaAct_Izq := "DB900_Estado_Mesas".EstadoVI[#OrdenEnCurso.EnH02_MesaDesCarga].Etapas_Carga_E1 OR
                   "DB900_Estado_Mesas".EstadoVI[#OrdenEnCurso.EnH02_MesaDesCarga].Etapas_Carga_E2 OR
                   "DB900_Estado_Mesas".EstadoVI[#OrdenEnCurso.EnH02_MesaDesCarga].Etapas_Carga_E3 OR
                   "DB900_Estado_Mesas".EstadoVI[#OrdenEnCurso.EnH02_MesaDesCarga].Etapas_Carga_E4;
               END_IF;

           END_IF;
       END_IF;


   END_IF;
END_REGION

REGION Network 33: >>>>>>>>>>>>>>>>>>>>>>>>>>>>>>>>>>>>>>>>>>>>>>>>>>>>>>>>>>>>>>>>>>>>>>>>>>>>>>>>
END_REGION

REGION Network 34: PETICION DE POSICIONAMIENTO >>> Calculo de la Orden para el Variador i950
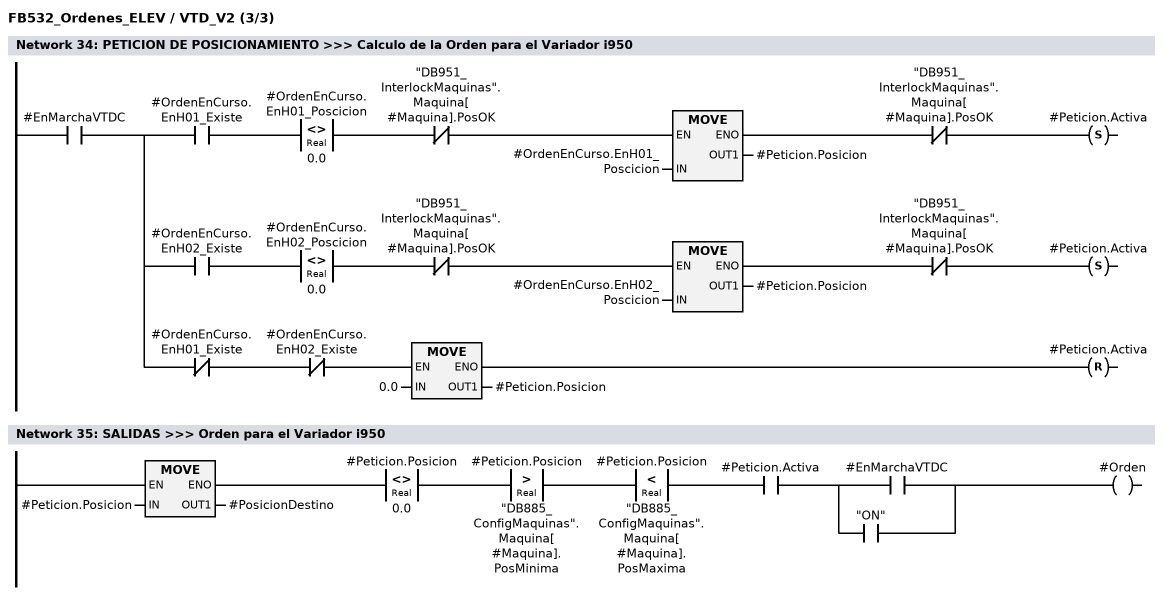
   RUNG wire#powerrail
      Contact( #EnMarchaVTDC )
      wire#w1
      Contact( #OrdenEnCurso.EnH01_Existe )
      { S7_Templates := "SrcType := Real" } NE_Contact(in1 := #OrdenEnCurso.EnH01_Poscicion, in2 := 0.0)
      I_Contact( "DB951_InterlockMaquinas".Maquina[#Maquina].PosOK )
      Move(in := #OrdenEnCurso.EnH01_Poscicion, out1 => #Peticion.Posicion)
      I_Contact( "DB951_InterlockMaquinas".Maquina[#Maquina].PosOK )
      S_Coil( #Peticion.Activa )
   END_RUNG
   RUNG wire#w1
      Contact( #OrdenEnCurso.EnH02_Existe )
      { S7_Templates := "SrcType := Real" } NE_Contact(in1 := #OrdenEnCurso.EnH02_Poscicion, in2 := 0.0)
      I_Contact( "DB951_InterlockMaquinas".Maquina[#Maquina].PosOK )
      Move(in := #OrdenEnCurso.EnH02_Poscicion, out1 => #Peticion.Posicion)
      I_Contact( "DB951_InterlockMaquinas".Maquina[#Maquina].PosOK )
      S_Coil( #Peticion.Activa )
   END_RUNG
   RUNG wire#w1
      I_Contact( #OrdenEnCurso.EnH01_Existe )
      I_Contact( #OrdenEnCurso.EnH02_Existe )
      Move(in := 0.0, out1 => #Peticion.Posicion)
      R_Coil( #Peticion.Activa )
   END_RUNG
   // the same network as SCL:
   #_w1 := #EnMarchaVTDC AND #OrdenEnCurso.EnH01_Existe AND (#OrdenEnCurso.EnH01_Poscicion <> 0.0) AND NOT "DB951_InterlockMaquinas".Maquina[#Maquina].PosOK;
   IF #_w1 THEN #Peticion.Posicion := #OrdenEnCurso.EnH01_Poscicion; END_IF;
   IF #_w1 AND NOT "DB951_InterlockMaquinas".Maquina[#Maquina].PosOK THEN #Peticion.Activa := TRUE; END_IF;
   #_w2 := #EnMarchaVTDC AND #OrdenEnCurso.EnH02_Existe AND (#OrdenEnCurso.EnH02_Poscicion <> 0.0) AND NOT "DB951_InterlockMaquinas".Maquina[#Maquina].PosOK;
   IF #_w2 THEN #Peticion.Posicion := #OrdenEnCurso.EnH02_Poscicion; END_IF;
   IF #_w2 AND NOT "DB951_InterlockMaquinas".Maquina[#Maquina].PosOK THEN #Peticion.Activa := TRUE; END_IF;
   IF #EnMarchaVTDC AND NOT #OrdenEnCurso.EnH01_Existe AND NOT #OrdenEnCurso.EnH02_Existe THEN
       #Peticion.Posicion := 0.0;
       #Peticion.Activa := FALSE;
   END_IF;
END_REGION

REGION Network 35: SALIDAS >>> Orden para el Variador i950
   RUNG wire#powerrail
      Move(in := #Peticion.Posicion, out1 => #PosicionDestino)
      { S7_Templates := "SrcType := Real" } NE_Contact(in1 := #Peticion.Posicion, in2 := 0.0)
      { S7_Templates := "SrcType := Real" } GT_Contact(in1 := #Peticion.Posicion, in2 := "DB885_ConfigMaquinas".Maquina[#Maquina].PosMinima)
      { S7_Templates := "SrcType := Real" } LT_Contact(in1 := #Peticion.Posicion, in2 := "DB885_ConfigMaquinas".Maquina[#Maquina].PosMaxima)
      Contact( #Peticion.Activa )
      wire#w1
      Contact( #EnMarchaVTDC )
      wire#w2
      Coil( #Orden )
   END_RUNG
   RUNG wire#w1
      Contact( "ON" )
   END_RUNG wire#w2
   // the same network as SCL:
   #PosicionDestino := #Peticion.Posicion;
   #Orden := (#Peticion.Posicion <> 0.0) AND (#Peticion.Posicion > "DB885_ConfigMaquinas".Maquina[#Maquina].PosMinima) AND (#Peticion.Posicion < "DB885_ConfigMaquinas".Maquina[#Maquina].PosMaxima) AND #Peticion.Activa AND (#EnMarchaVTDC OR "ON");
END_REGION

REGION Network 36: >>>>>>>>>>>>>>>>>>>>>>>>>>>>>>>>>>>>>>>>>>>>>>>>>>>>>>>>>>>>>>>>>>>>>>>>>>>>>>>>
END_REGION
END_FUNCTION_BLOCK
